KUKA KRL program: EPS_2_251455_MH11A_A_20251003045056.src

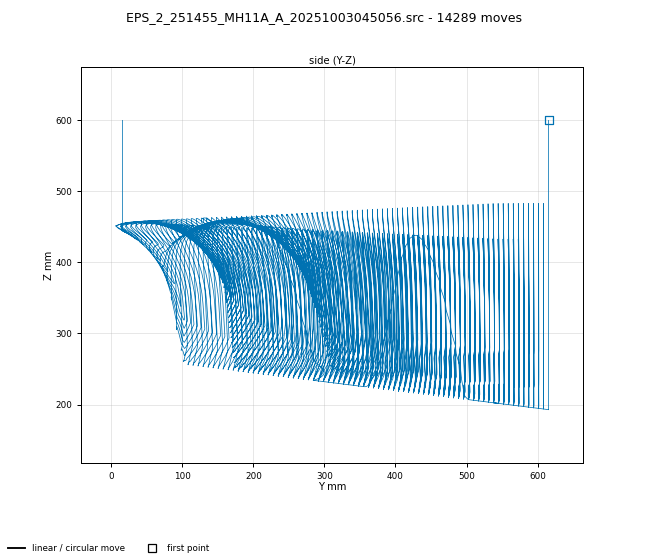
[picture p0: tool path of EPS_2_251455_MH11A_A_20251003045056.src, 14289 of 14291 moves have a stored position in this frame; points joined in program order, loops and branches not executed]
&ACCESS RVP
&REL 4
&COMMENT QRS 19112012
&PARAM EDITMASK = *
DEF PART()
EXT BAS (BAS_COMMAND :IN,REAL :IN )
INT I
BAS (#INITMOV,0 )

;KUKA QRS Post kuka4.cps  Date:22-06-2017 !

File_ID=2867

QRS_PRE_INIT()

;Init var - Until changes are made in qrs_pre_init
Outlet_Square_prg=0
Inlet_1_Square_prg=0
Inlet_2_Square_prg=0
Inlet_3_Square_prg=0
Inlet_4_Square_prg=0
Inlet_5_Square_prg=0

Outlet_1={X 0.000, Y 540.910, Z 382.500, B 0.000, E1 0.000 }
Inlet_1={X 0.000, Y 544.470, Z 332.500, B 0.000, E1 166.000 }
Inlet_2={X 0.000, Y 544.470, Z 332.500, B 0.000, E1 269.000 }
Outlet_1_type=201
Inlet_1_type=201
Inlet_2_type=201
;QRS#1=Sidecore dimensions
;QRS#2=200-8" PVC SDR 35
;QRS#3=200-8" PVC SDR 35
;QRS#4=200-8" PVC SDR 35
;QRS#5=
;QRS#6=
;QRS#7=
;QRS#8=
;QRS#9=12-08 PSX
;QRS#10=12-08 PSX
;QRS#11=12-08 PSX
;QRS#12=
;QRS#13=
;QRS#14=
;QRS#15=
;QRS#16=1220x127x762 2,5'
;QRS#17=EPS Height
;QRS#18=483
;QRS#19=*
;QRS#20= UPDATED VERSION 22-06-2017
;QRS#21=*
Outlet_Square=0100
Inlet_1_Square=0100
Inlet_2_Square=0100
Inlet_3_Square=0
Inlet_4_Square=0
Inlet_5_Square=0
Mill_Square=1
Outlet_Square_Prg=204
Inlet_1_Square_prg=204
Inlet_2_Square_prg=204

QRS_INIT()

$ADVANCE=5

; T1
PTP {E1 173.609,E2 173.609}
PTP {X 0,Y 615.501,A -85,B 0,C 180,E1 173.609,E2 173.609,E3 0,E4 0,E5 0,E6 0}
QRS_SPEED_INIT()
LIN {X 0,Y 615.501,Z 600,A -85,B 0,C 180,E1 173.609,E2 173.609,E3 0,E4 0,E5 0,E6 0} C_VEL
LIN {X 0,Y 615.501,Z 202.87,A -85,B 0,C 180,E1 173.609,E2 173.609} C_VEL
LIN {X 0,Y 615.501,Z 194.691,A -85,B 0,C 180,E1 173.609,E2 173.609} C_VEL
LIN {X 0,Y 615.475,Z 192.691,A -85,B 0,C 180,E1 173.423,E2 173.423} C_VEL
LIN {X 0,Y 615.439,Z 192.695,A -85,B 0,C 180,E1 170.8,E2 170.8} C_VEL
LIN {X 0,Y 615.484,Z 192.701,A -85,B 0,C 180,E1 168.139,E2 168.139} C_VEL
LIN {X 0,Y 615.466,Z 192.69,A -85,B 0,C 180,E1 165.45,E2 165.45} C_VEL
LIN {X 0,Y 615.461,Z 192.69,A -85,B 0,C 180,E1 163.412,E2 163.412} C_VEL
LIN {X 0,Y 615.456,Z 192.69,A -85,B 0,C 180,E1 161.353,E2 161.353} C_VEL
LIN {X 0,Y 615.451,Z 192.691,A -85,B 0,C 180,E1 159.268,E2 159.268} C_VEL
LIN {X 0,Y 615.451,Z 192.692,A -85,B 0,C 180,E1 157.154,E2 157.154} C_VEL
LIN {X 0,Y 615.498,Z 192.699,A -85,B 0,C 180,E1 154.427,E2 154.427} C_VEL
LIN {X 0,Y 615.463,Z 192.689,A -85,B 0,C 180,E1 151.552,E2 151.552} C_VEL
LIN {X 0,Y 615.472,Z 192.697,A -85,B 0,C 180,E1 148.915,E2 148.915} C_VEL
LIN {X 0,Y 615.486,Z 192.685,A -85,B 0,C 180,E1 145.978,E2 145.978} C_VEL
LIN {X 0,Y 615.462,Z 192.689,A -85,B 0,C 180,E1 143.573,E2 143.573} C_VEL
LIN {X 0,Y 615.492,Z 192.699,A -85,B 0,C 180,E1 140.936,E2 140.936} C_VEL
LIN {X 0,Y 615.476,Z 192.686,A -85,B 0,C 180,E1 137.92,E2 137.92} C_VEL
LIN {X 0,Y 615.496,Z 192.699,A -85,B 0,C 180,E1 135.066,E2 135.066} C_VEL
LIN {X 0,Y 615.481,Z 192.684,A -85,B 0,C 180,E1 132.079,E2 132.079} C_VEL
LIN {X 0,Y 615.47,Z 192.691,A -85,B 0,C 180,E1 129.75,E2 129.75} C_VEL
LIN {X 0,Y 615.484,Z 192.693,A -85,B 0,C 180,E1 126.935,E2 126.935} C_VEL
LIN {X 0,Y 615.473,Z 192.688,A -85,B 0,C 180,E1 124.022,E2 124.022} C_VEL
LIN {X 0,Y 615.475,Z 192.815,A -85,B 0,C 180,E1 121.967,E2 121.967} C_VEL
LIN {X 0,Y 615.473,Z 207.433,A -85,B 0,C 180,E1 119.406,E2 119.406} C_VEL
LIN {X 0,Y 615.47,Z 222.393,A -85,B 0,C 180,E1 116.814,E2 116.814} C_VEL
LIN {X 0,Y 615.432,Z 328.155,A -85,B 0,C 180,E1 115.557,E2 115.557} C_VEL
LIN {X 0,Y 615.439,Z 341.34,A -85,B 0,C 180,E1 115.274,E2 115.274} C_VEL
LIN {X 0,Y 615.476,Z 354.247,A -85,B 0,C 180,E1 114.856,E2 114.856} C_VEL
LIN {X 0,Y 615.479,Z 365.558,A -85,B 0,C 180,E1 114.361,E2 114.361} C_VEL
LIN {X 0,Y 615.469,Z 376.031,A -85,B 0,C 180,E1 113.779,E2 113.779} C_VEL
LIN {X 0,Y 615.498,Z 386.868,A -85,B 0,C 180,E1 113.021,E2 113.021} C_VEL
LIN {X 0,Y 615.498,Z 397.085,A -85,B 0,C 180,E1 112.135,E2 112.135} C_VEL
LIN {X 0,Y 615.497,Z 405.273,A -85,B 0,C 180,E1 111.255,E2 111.255} C_VEL
LIN {X 0,Y 615.496,Z 412.557,A -85,B 0,C 180,E1 110.295,E2 110.295} C_VEL
LIN {X 0,Y 615.497,Z 418.434,A -85,B 0,C 180,E1 109.337,E2 109.337} C_VEL
LIN {X 0,Y 615.496,Z 423.553,A -85,B 0,C 180,E1 108.281,E2 108.281} C_VEL
LIN {X 0,Y 615.498,Z 427.265,A -85,B 0,C 180,E1 107.269,E2 107.269} C_VEL
LIN {X 0,Y 615.495,Z 429.552,A -85,B 0,C 180,E1 106.432,E2 106.432} C_VEL
LIN {X 0,Y 615.496,Z 431.625,A -85,B 0,C 180,E1 105.225,E2 105.225} C_VEL
LIN {X 0,Y 615.499,Z 432.387,A -85,B 0,C 180,E1 103.935,E2 103.935} C_VEL
LIN {X 0,Y 615.496,Z 432.102,A -85,B 0,C 180,E1 103.2,E2 103.2} C_VEL
LIN {X 0,Y 615.496,Z 431.442,A -85,B 0,C 180,E1 102.529,E2 102.529} C_VEL
LIN {X 0,Y 615.494,Z 430.377,A -85,B 0,C 180,E1 101.86,E2 101.86} C_VEL
LIN {X 0,Y 615.495,Z 428.034,A -85,B 0,C 180,E1 100.889,E2 100.889} C_VEL
LIN {X 0,Y 615.498,Z 424.523,A -85,B 0,C 180,E1 99.861,E2 99.861} C_VEL
LIN {X 0,Y 615.498,Z 420.016,A -85,B 0,C 180,E1 98.867,E2 98.867} C_VEL
LIN {X 0,Y 615.499,Z 413.193,A -85,B 0,C 180,E1 97.71,E2 97.71} C_VEL
LIN {X 0,Y 615.498,Z 405.966,A -85,B 0,C 180,E1 96.74,E2 96.74} C_VEL
LIN {X 0,Y 615.499,Z 398.311,A -85,B 0,C 180,E1 95.898,E2 95.898} C_VEL
LIN {X 0,Y 615.498,Z 389.248,A -85,B 0,C 180,E1 95.076,E2 95.076} C_VEL
LIN {X 0,Y 615.477,Z 379.211,A -85,B 0,C 180,E1 94.338,E2 94.338} C_VEL
LIN {X 0,Y 615.462,Z 368.138,A -85,B 0,C 180,E1 93.682,E2 93.682} C_VEL
LIN {X 0,Y 615.496,Z 357.647,A -85,B 0,C 180,E1 93.19,E2 93.19} C_VEL
LIN {X 0,Y 615.477,Z 345.076,A -85,B 0,C 180,E1 92.74,E2 92.74} C_VEL
LIN {X 0,Y 615.457,Z 332.551,A -85,B 0,C 180,E1 92.433,E2 92.433} C_VEL
LIN {X 0,Y 615.454,Z 314.913,A -85,B 0,C 180,E1 92.188,E2 92.188} C_VEL
LIN {X 0,Y 615.495,Z 222.43,A -85,B 0,C 180,E1 91.103,E2 91.103} C_VEL
LIN {X 0,Y 615.488,Z 206.621,A -85,B 0,C 180,E1 88.363,E2 88.363} C_VEL
LIN {X 0,Y 615.455,Z 192.693,A -85,B 0,C 180,E1 85.907,E2 85.907} C_VEL
LIN {X 0,Y 615.467,Z 192.688,A -85,B 0,C 180,E1 83.442,E2 83.442} C_VEL
LIN {X 0,Y 615.495,Z 192.696,A -85,B 0,C 180,E1 80.801,E2 80.801} C_VEL
LIN {X 0,Y 615.451,Z 192.695,A -85,B 0,C 180,E1 78.138,E2 78.138} C_VEL
LIN {X 0,Y 615.444,Z 192.695,A -85,B 0,C 180,E1 76.086,E2 76.086} C_VEL
LIN {X 0,Y 615.483,Z 192.688,A -85,B 0,C 180,E1 73.413,E2 73.413} C_VEL
LIN {X 0,Y 615.467,Z 192.698,A -85,B 0,C 180,E1 70.661,E2 70.661} C_VEL
LIN {X 0,Y 615.454,Z 192.697,A -85,B 0,C 180,E1 68.566,E2 68.566} C_VEL
LIN {X 0,Y 615.443,Z 192.693,A -85,B 0,C 180,E1 66.002,E2 66.002} C_VEL
LIN {X 0,Y 615.479,Z 192.692,A -85,B 0,C 180,E1 63.555,E2 63.555} C_VEL
LIN {X 0,Y 615.493,Z 192.697,A -85,B 0,C 180,E1 61.342,E2 61.342} C_VEL
LIN {X 0,Y 615.456,Z 192.698,A -85,B 0,C 180,E1 58.92,E2 58.92} C_VEL
LIN {X 0,Y 615.429,Z 192.697,A -85,B 0,C 180,E1 56.475,E2 56.475} C_VEL
LIN {X 0,Y 615.437,Z 192.695,A -85,B 0,C 180,E1 54.174,E2 54.174} C_VEL
LIN {X 0,Y 615.46,Z 192.695,A -85,B 0,C 180,E1 51.929,E2 51.929} C_VEL
LIN {X 0,Y 615.478,Z 192.7,A -85,B 0,C 180,E1 49.392,E2 49.392} C_VEL
LIN {X 0,Y 615.428,Z 192.699,A -85,B 0,C 180,E1 46.959,E2 46.959} C_VEL
LIN {X 0,Y 615.422,Z 192.699,A -85,B 0,C 180,E1 44.925,E2 44.925} C_VEL
LIN {X 0,Y 615.459,Z 192.698,A -85,B 0,C 180,E1 42.076,E2 42.076} C_VEL
LIN {X 0,Y 615.484,Z 192.701,A -85,B 0,C 180,E1 39.751,E2 39.751} C_VEL
LIN {X 0,Y 615.423,Z 192.7,A -85,B 0,C 180,E1 37.247,E2 37.247} C_VEL
LIN {X 0,Y 615.455,Z 192.7,A -85,B 0,C 180,E1 35.618,E2 35.618} C_VEL
LIN {X 0,Y 615.422,Z 192.699,A -85,B 0,C 180,E1 33.241,E2 33.241} C_VEL
LIN {X 0,Y 615.418,Z 192.699,A -85,B 0,C 180,E1 30.924,E2 30.924} C_VEL
LIN {X 0,Y 615.457,Z 192.699,A -85,B 0,C 180,E1 28.444,E2 28.444} C_VEL
LIN {X 0,Y 615.439,Z 192.696,A -85,B 0,C 180,E1 25.558,E2 25.558} C_VEL
LIN {X 0,Y 615.438,Z 192.696,A -85,B 0,C 180,E1 23.559,E2 23.559} C_VEL
LIN {X 0,Y 615.431,Z 192.696,A -85,B 0,C 180,E1 21.434,E2 21.434} C_VEL
LIN {X 0,Y 615.439,Z 192.798,A -85,B 0,C 180,E1 18.972,E2 18.972} C_VEL
LIN {X 0,Y 615.49,Z 208.798,A -85,B 0,C 180,E1 16.168,E2 16.168} C_VEL
LIN {X 0,Y 615.482,Z 222.406,A -85,B 0,C 180,E1 13.811,E2 13.811} C_VEL
LIN {X 0,Y 615.482,Z 329.594,A -85,B 0,C 180,E1 12.53,E2 12.53} C_VEL
LIN {X 0,Y 615.496,Z 342.645,A -85,B 0,C 180,E1 12.237,E2 12.237} C_VEL
LIN {X 0,Y 615.494,Z 355.228,A -85,B 0,C 180,E1 11.819,E2 11.819} C_VEL
LIN {X 0,Y 615.465,Z 367.214,A -85,B 0,C 180,E1 11.277,E2 11.277} C_VEL
LIN {X 0,Y 615.476,Z 378.576,A -85,B 0,C 180,E1 10.614,E2 10.614} C_VEL
LIN {X 0,Y 615.499,Z 388.888,A -85,B 0,C 180,E1 9.862,E2 9.862} C_VEL
LIN {X 0,Y 615.497,Z 398.107,A -85,B 0,C 180,E1 9.033,E2 9.033} C_VEL
LIN {X 0,Y 615.498,Z 407.028,A -85,B 0,C 180,E1 8.041,E2 8.041} C_VEL
LIN {X 0,Y 615.497,Z 414.162,A -85,B 0,C 180,E1 7.057,E2 7.057} C_VEL
LIN {X 0,Y 615.498,Z 419.032,A -85,B 0,C 180,E1 6.228,E2 6.228} C_VEL
LIN {X 0,Y 615.495,Z 423.722,A -85,B 0,C 180,E1 5.241,E2 5.241} C_VEL
LIN {X 0,Y 615.496,Z 427.306,A -85,B 0,C 180,E1 4.257,E2 4.257} C_VEL
LIN {X 0,Y 615.496,Z 429.894,A -85,B 0,C 180,E1 3.273,E2 3.273} C_VEL
LIN {X 0,Y 615.497,Z 431.108,A -85,B 0,C 180,E1 2.618,E2 2.618} C_VEL
LIN {X 0,Y 615.496,Z 431.923,A -85,B 0,C 180,E1 1.963,E2 1.963} C_VEL
LIN {X 0,Y 615.495,Z 432.323,A -85,B 0,C 180,E1 0.654,E2 0.654} C_VEL
LIN {X 0,Y 615.495,Z 431.962,A -85,B 0,C 180,E1 0,E2 0} C_VEL
LIN {X 0,Y 615.496,Z 431.198,A -85,B 0,C 180,E1 -0.654,E2 -0.654} C_VEL
LIN {X 0,Y 615.499,Z 428.43,A -85,B 0,C 180,E1 -1.963,E2 -1.963} C_VEL
LIN {X 0,Y 615.496,Z 425.246,A -85,B 0,C 180,E1 -2.945,E2 -2.945} C_VEL
LIN {X 0,Y 615.495,Z 421.016,A -85,B 0,C 180,E1 -3.928,E2 -3.928} C_VEL
LIN {X 0,Y 615.497,Z 414.61,A -85,B 0,C 180,E1 -5.077,E2 -5.077} C_VEL
LIN {X 0,Y 615.497,Z 407.586,A -85,B 0,C 180,E1 -6.063,E2 -6.063} C_VEL
LIN {X 0,Y 615.498,Z 398.755,A -85,B 0,C 180,E1 -7.057,E2 -7.057} C_VEL
LIN {X 0,Y 615.497,Z 389.831,A -85,B 0,C 180,E1 -7.875,E2 -7.875} C_VEL
LIN {X 0,Y 615.489,Z 379.866,A -85,B 0,C 180,E1 -8.619,E2 -8.619} C_VEL
LIN {X 0,Y 615.492,Z 368.809,A -85,B 0,C 180,E1 -9.281,E2 -9.281} C_VEL
LIN {X 0,Y 615.489,Z 356.416,A -85,B 0,C 180,E1 -9.862,E2 -9.862} C_VEL
LIN {X 0,Y 615.452,Z 344.471,A -85,B 0,C 180,E1 -10.278,E2 -10.278} C_VEL
LIN {X 0,Y 615.446,Z 331.21,A -85,B 0,C 180,E1 -10.592,E2 -10.592} C_VEL
LIN {X 0,Y 615.455,Z 309.997,A -85,B 0,C 180,E1 -10.87,E2 -10.87} C_VEL
LIN {X 0,Y 615.449,Z 222.404,A -85,B 0,C 180,E1 -11.903,E2 -11.903} C_VEL
LIN {X 0,Y 615.447,Z 208.959,A -85,B 0,C 180,E1 -14.232,E2 -14.232} C_VEL
LIN {X 0,Y 615.489,Z 193.058,A -85,B 0,C 180,E1 -17.014,E2 -17.014} C_VEL
LIN {X 0,Y 615.488,Z 192.686,A -85,B 0,C 180,E1 -17.099,E2 -17.099} C_VEL
LIN {X 0,Y 615.483,Z 192.684,A -85,B 0,C 180,E1 -19.338,E2 -19.338} C_VEL
LIN {X 0,Y 615.472,Z 192.696,A -85,B 0,C 180,E1 -22.137,E2 -22.137} C_VEL
LIN {X 0,Y 615.495,Z 192.684,A -85,B 0,C 180,E1 -24.991,E2 -24.991} C_VEL
LIN {X 0,Y 615.486,Z 192.683,A -85,B 0,C 180,E1 -27.177,E2 -27.177} C_VEL
LIN {X 0,Y 615.463,Z 192.693,A -85,B 0,C 180,E1 -29.79,E2 -29.79} C_VEL
LIN {X 0,Y 615.49,Z 192.696,A -85,B 0,C 180,E1 -32.457,E2 -32.457} C_VEL
LIN {X 0,Y 615.493,Z 192.685,A -85,B 0,C 180,E1 -34.815,E2 -34.815} C_VEL
LIN {X 0,Y 615.468,Z 192.687,A -85,B 0,C 180,E1 -37.244,E2 -37.244} C_VEL
LIN {X 0,Y 615.491,Z 192.699,A -85,B 0,C 180,E1 -40.089,E2 -40.089} C_VEL
LIN {X 0,Y 615.475,Z 192.685,A -85,B 0,C 180,E1 -43.045,E2 -43.045} C_VEL
LIN {X 0,Y 615.476,Z 192.697,A -85,B 0,C 180,E1 -45.849,E2 -45.849} C_VEL
LIN {X 0,Y 615.493,Z 192.687,A -85,B 0,C 180,E1 -48.526,E2 -48.526} C_VEL
LIN {X 0,Y 615.463,Z 192.688,A -85,B 0,C 180,E1 -51.093,E2 -51.093} C_VEL
LIN {X 0,Y 615.465,Z 192.695,A -85,B 0,C 180,E1 -53.573,E2 -53.573} C_VEL
LIN {X 0,Y 615.495,Z 192.685,A -85,B 0,C 180,E1 -56.465,E2 -56.465} C_VEL
LIN {X 0,Y 615.459,Z 192.69,A -85,B 0,C 180,E1 -59.078,E2 -59.078} C_VEL
LIN {X 0,Y 615.47,Z 192.696,A -85,B 0,C 180,E1 -61.553,E2 -61.553} C_VEL
LIN {X 0,Y 615.498,Z 192.683,A -85,B 0,C 180,E1 -64.43,E2 -64.43} C_VEL
LIN {X 0,Y 615.456,Z 192.818,A -85,B 0,C 180,E1 -67.065,E2 -67.065} C_VEL
LIN {X 0,Y 615.471,Z 212.766,A -85,B 0,C 180,E1 -69.706,E2 -69.706} C_VEL
LIN {X 0,Y 615.477,Z 234.665,A -85,B 0,C 180,E1 -72.557,E2 -72.557} C_VEL
LIN {X 0,Y 615.471,Z 255.886,A -85,B 0,C 180,E1 -75.281,E2 -75.281} C_VEL
LIN {X 0,Y 615.452,Z 270.295,A -85,B 0,C 180,E1 -77.112,E2 -77.112} C_VEL
LIN {X 0,Y 615.483,Z 378.793,A -85,B 0,C 180,E1 -78.41,E2 -78.41} C_VEL
LIN {X 0,Y 615.474,Z 391.321,A -85,B 0,C 180,E1 -78.681,E2 -78.681} C_VEL
LIN {X 0,Y 615.487,Z 404.628,A -85,B 0,C 180,E1 -79.113,E2 -79.113} C_VEL
LIN {X 0,Y 615.479,Z 416.465,A -85,B 0,C 180,E1 -79.639,E2 -79.639} C_VEL
LIN {X 0,Y 615.496,Z 427.983,A -85,B 0,C 180,E1 -80.303,E2 -80.303} C_VEL
LIN {X 0,Y 615.499,Z 438.332,A -85,B 0,C 180,E1 -81.049,E2 -81.049} C_VEL
LIN {X 0,Y 615.497,Z 446.804,A -85,B 0,C 180,E1 -81.793,E2 -81.793} C_VEL
LIN {X 0,Y 615.498,Z 454.6,A -85,B 0,C 180,E1 -82.619,E2 -82.619} C_VEL
LIN {X 0,Y 615.496,Z 462.198,A -85,B 0,C 180,E1 -83.607,E2 -83.607} C_VEL
LIN {X 0,Y 615.498,Z 469.201,A -85,B 0,C 180,E1 -84.758,E2 -84.758} C_VEL
LIN {X 0,Y 615.494,Z 473.848,A -85,B 0,C 180,E1 -85.743,E2 -85.743} C_VEL
LIN {X 0,Y 615.494,Z 477.396,A -85,B 0,C 180,E1 -86.726,E2 -86.726} C_VEL
LIN {X 0,Y 615.497,Z 479.231,A -85,B 0,C 180,E1 -87.381,E2 -87.381} C_VEL
LIN {X 0,Y 615.5,Z 480.606,A -85,B 0,C 180,E1 -88.036,E2 -88.036} C_VEL
LIN {X 0,Y 615.496,Z 482.173,A -85,B 0,C 180,E1 -89.345,E2 -89.345} C_VEL
LIN {X 0,Y 615.494,Z 482.389,A -85,B 0,C 180,E1 -89.999,E2 -89.999} C_VEL
LIN {X 0,Y 615.495,Z 481.581,A -85,B 0,C 180,E1 -91.308,E2 -91.308} C_VEL
LIN {X 0,Y 615.5,Z 480.609,A -85,B 0,C 180,E1 -91.962,E2 -91.962} C_VEL
LIN {X 0,Y 615.497,Z 479.235,A -85,B 0,C 180,E1 -92.617,E2 -92.617} C_VEL
LIN {X 0,Y 615.496,Z 476.352,A -85,B 0,C 180,E1 -93.6,E2 -93.6} C_VEL
LIN {X 0,Y 615.498,Z 472.445,A -85,B 0,C 180,E1 -94.584,E2 -94.584} C_VEL
LIN {X 0,Y 615.499,Z 467.409,A -85,B 0,C 180,E1 -95.569,E2 -95.569} C_VEL
LIN {X 0,Y 615.497,Z 460.869,A -85,B 0,C 180,E1 -96.583,E2 -96.583} C_VEL
LIN {X 0,Y 615.497,Z 453.14,A -85,B 0,C 180,E1 -97.545,E2 -97.545} C_VEL
LIN {X 0,Y 615.498,Z 445.053,A -85,B 0,C 180,E1 -98.37,E2 -98.37} C_VEL
LIN {X 0,Y 615.499,Z 435.178,A -85,B 0,C 180,E1 -99.198,E2 -99.198} C_VEL
LIN {X 0,Y 615.492,Z 423.994,A -85,B 0,C 180,E1 -99.944,E2 -99.944} C_VEL
LIN {X 0,Y 615.483,Z 413.039,A -85,B 0,C 180,E1 -100.526,E2 -100.526} C_VEL
LIN {X 0,Y 615.478,Z 400.507,A -85,B 0,C 180,E1 -101.04,E2 -101.04} C_VEL
LIN {X 0,Y 615.475,Z 388.102,A -85,B 0,C 180,E1 -101.401,E2 -101.401} C_VEL
LIN {X 0,Y 615.487,Z 374.523,A -85,B 0,C 180,E1 -101.651,E2 -101.651} C_VEL
LIN {X 0,Y 615.452,Z 270.307,A -85,B 0,C 180,E1 -102.886,E2 -102.886} C_VEL
LIN {X 0,Y 615.498,Z 247.939,A -85,B 0,C 180,E1 -105.734,E2 -105.734} C_VEL
LIN {X 0,Y 615.452,Z 225.786,A -85,B 0,C 180,E1 -108.594,E2 -108.594} C_VEL
LIN {X 0,Y 615.484,Z 205.459,A -85,B 0,C 180,E1 -111.256,E2 -111.256} C_VEL
LIN {X 0,Y 615.456,Z 192.691,A -85,B 0,C 180,E1 -112.978,E2 -112.978} C_VEL
LIN {X 0,Y 615.493,Z 192.689,A -85,B 0,C 180,E1 -115.715,E2 -115.715} C_VEL
LIN {X 0,Y 615.453,Z 192.694,A -85,B 0,C 180,E1 -118.659,E2 -118.659} C_VEL
LIN {X 0,Y 615.461,Z 192.689,A -85,B 0,C 180,E1 -121.081,E2 -121.081} C_VEL
LIN {X 0,Y 615.481,Z 192.7,A -85,B 0,C 180,E1 -124.021,E2 -124.021} C_VEL
LIN {X 0,Y 615.448,Z 192.695,A -85,B 0,C 180,E1 -126.426,E2 -126.426} C_VEL
LIN {X 0,Y 615.466,Z 192.69,A -85,B 0,C 180,E1 -129.059,E2 -129.059} C_VEL
LIN {X 0,Y 615.494,Z 192.694,A -85,B 0,C 180,E1 -131.472,E2 -131.472} C_VEL
LIN {X 0,Y 615.445,Z 192.697,A -85,B 0,C 180,E1 -134.152,E2 -134.152} C_VEL
LIN {X 0,Y 615.467,Z 192.692,A -85,B 0,C 180,E1 -136.953,E2 -136.953} C_VEL
LIN {X 0,Y 615.446,Z 192.698,A -85,B 0,C 180,E1 -139.914,E2 -139.914} C_VEL
LIN {X 0,Y 615.434,Z 192.698,A -85,B 0,C 180,E1 -141.993,E2 -141.993} C_VEL
LIN {X 0,Y 615.432,Z 192.696,A -85,B 0,C 180,E1 -144.38,E2 -144.38} C_VEL
LIN {X 0,Y 615.461,Z 192.695,A -85,B 0,C 180,E1 -146.762,E2 -146.762} C_VEL
LIN {X 0,Y 615.492,Z 192.699,A -85,B 0,C 180,E1 -149.08,E2 -149.08} C_VEL
LIN {X 0,Y 615.442,Z 192.699,A -85,B 0,C 180,E1 -151.556,E2 -151.556} C_VEL
LIN {X 0,Y 615.435,Z 192.7,A -85,B 0,C 180,E1 -153.553,E2 -153.553} C_VEL
LIN {X 0,Y 615.421,Z 192.699,A -85,B 0,C 180,E1 -155.725,E2 -155.725} C_VEL
LIN {X 0,Y 615.413,Z 192.7,A -85,B 0,C 180,E1 -157.861,E2 -157.861} C_VEL
LIN {X 0,Y 615.474,Z 192.7,A -85,B 0,C 180,E1 -160.662,E2 -160.662} C_VEL
LIN {X 0,Y 615.424,Z 192.7,A -85,B 0,C 180,E1 -163.412,E2 -163.412} C_VEL
LIN {X 0,Y 615.422,Z 192.699,A -85,B 0,C 180,E1 -165.449,E2 -165.449} C_VEL
LIN {X 0,Y 615.42,Z 192.699,A -85,B 0,C 180,E1 -167.469,E2 -167.469} C_VEL
LIN {X 0,Y 615.422,Z 192.698,A -85,B 0,C 180,E1 -169.472,E2 -169.472} C_VEL
LIN {X 0,Y 615.423,Z 192.698,A -85,B 0,C 180,E1 -171.463,E2 -171.463} C_VEL
LIN {X 0,Y 615.454,Z 192.699,A -85,B 0,C 180,E1 -174.101,E2 -174.101} C_VEL
LIN {X 0,Y 615.473,Z 192.694,A -85,B 0,C 180,E1 -176.727,E2 -176.727} C_VEL
LIN {X 0,Y 615.43,Z 192.696,A -85,B 0,C 180,E1 -179.346,E2 -179.346} C_VEL
LIN {X 0,Y 615.467,Z 192.699,A -85,B 0,C 180,E1 -181.963,E2 -181.963} C_VEL
LIN {X 0,Y 615.478,Z 192.691,A -85,B 0,C 180,E1 -184.585,E2 -184.585} C_VEL
LIN {X 0,Y 615.475,Z 192.691,A -85,B 0,C 180,E1 -186.577,E2 -186.577} C_VEL
LIN {X 0,Y 614.772,Z 192.839,A -85,B 0,C 180,E1 -187.123,E2 -187.123} C_VEL
LIN {X 0,Y 611.916,Z 193.266,A -85,B 0,C 180,E1 -188.009,E2 -188.009} C_VEL
LIN {X 0,Y 609.53,Z 193.569,A -85,B 0,C 180,E1 -188.721,E2 -188.721} C_VEL
LIN {X 0,Y 608.51,Z 193.683,A -85,B 0,C 180,E1 -189.271,E2 -189.271} C_VEL
LIN {X 0,Y 608.429,Z 193.693,A -85,B 0,C 180,E1 -189.457,E2 -189.457} C_VEL
LIN {X 0,Y 608.456,Z 193.696,A -85,B 0,C 180,E1 -192,E2 -192} C_VEL
LIN {X 0,Y 608.453,Z 193.688,A -85,B 0,C 180,E1 -194.721,E2 -194.721} C_VEL
LIN {X 0,Y 608.434,Z 193.695,A -85,B 0,C 180,E1 -197.477,E2 -197.477} C_VEL
LIN {X 0,Y 608.455,Z 193.689,A -85,B 0,C 180,E1 -200.275,E2 -200.275} C_VEL
LIN {X 0,Y 608.452,Z 193.688,A -85,B 0,C 180,E1 -202.477,E2 -202.477} C_VEL
LIN {X 0,Y 608.437,Z 193.689,A -85,B 0,C 180,E1 -204.572,E2 -204.572} C_VEL
LIN {X 0,Y 608.463,Z 193.692,A -85,B 0,C 180,E1 -207.206,E2 -207.206} C_VEL
LIN {X 0,Y 608.469,Z 193.687,A -85,B 0,C 180,E1 -209.974,E2 -209.974} C_VEL
LIN {X 0,Y 608.439,Z 193.69,A -85,B 0,C 180,E1 -212.521,E2 -212.521} C_VEL
LIN {X 0,Y 608.433,Z 193.694,A -85,B 0,C 180,E1 -214.905,E2 -214.905} C_VEL
LIN {X 0,Y 608.476,Z 193.695,A -85,B 0,C 180,E1 -217.161,E2 -217.161} C_VEL
LIN {X 0,Y 608.477,Z 193.69,A -85,B 0,C 180,E1 -219.44,E2 -219.44} C_VEL
LIN {X 0,Y 608.438,Z 193.69,A -85,B 0,C 180,E1 -222.333,E2 -222.333} C_VEL
LIN {X 0,Y 608.46,Z 193.694,A -85,B 0,C 180,E1 -224.796,E2 -224.796} C_VEL
LIN {X 0,Y 608.467,Z 193.686,A -85,B 0,C 180,E1 -227.666,E2 -227.666} C_VEL
LIN {X 0,Y 608.446,Z 193.697,A -85,B 0,C 180,E1 -230.706,E2 -230.706} C_VEL
LIN {X 0,Y 608.455,Z 193.692,A -85,B 0,C 180,E1 -233.086,E2 -233.086} C_VEL
LIN {X 0,Y 608.465,Z 193.686,A -85,B 0,C 180,E1 -235.532,E2 -235.532} C_VEL
LIN {X 0,Y 608.479,Z 193.809,A -85,B 0,C 180,E1 -237.981,E2 -237.981} C_VEL
LIN {X 0,Y 608.464,Z 208.651,A -85,B 0,C 180,E1 -240.602,E2 -240.602} C_VEL
LIN {X 0,Y 608.442,Z 222.619,A -85,B 0,C 180,E1 -243.039,E2 -243.039} C_VEL
LIN {X 0,Y 608.499,Z 329.351,A -85,B 0,C 180,E1 -244.328,E2 -244.328} C_VEL
LIN {X 0,Y 608.475,Z 342.727,A -85,B 0,C 180,E1 -244.63,E2 -244.63} C_VEL
LIN {X 0,Y 608.523,Z 355.714,A -85,B 0,C 180,E1 -245.069,E2 -245.069} C_VEL
LIN {X 0,Y 608.498,Z 367.699,A -85,B 0,C 180,E1 -245.621,E2 -245.621} C_VEL
LIN {X 0,Y 608.481,Z 379.741,A -85,B 0,C 180,E1 -246.337,E2 -246.337} C_VEL
LIN {X 0,Y 608.491,Z 390.515,A -85,B 0,C 180,E1 -247.148,E2 -247.148} C_VEL
LIN {X 0,Y 608.456,Z 399.194,A -85,B 0,C 180,E1 -247.952,E2 -247.952} C_VEL
LIN {X 0,Y 608.449,Z 407.117,A -85,B 0,C 180,E1 -248.842,E2 -248.842} C_VEL
LIN {X 0,Y 608.438,Z 414.789,A -85,B 0,C 180,E1 -249.902,E2 -249.902} C_VEL
LIN {X 0,Y 608.44,Z 419.887,A -85,B 0,C 180,E1 -250.781,E2 -250.781} C_VEL
LIN {X 0,Y 608.43,Z 424.752,A -85,B 0,C 180,E1 -251.828,E2 -251.828} C_VEL
LIN {X 0,Y 608.453,Z 428.39,A -85,B 0,C 180,E1 -252.871,E2 -252.871} C_VEL
LIN {X 0,Y 608.434,Z 430.925,A -85,B 0,C 180,E1 -253.906,E2 -253.906} C_VEL
LIN {X 0,Y 608.42,Z 432.034,A -85,B 0,C 180,E1 -254.594,E2 -254.594} C_VEL
LIN {X 0,Y 608.418,Z 432.71,A -85,B 0,C 180,E1 -255.279,E2 -255.279} C_VEL
LIN {X 0,Y 608.445,Z 432.994,A -85,B 0,C 180,E1 -255.995,E2 -255.995} C_VEL
LIN {X 0,Y 608.439,Z 432.828,A -85,B 0,C 180,E1 -256.644,E2 -256.644} C_VEL
LIN {X 0,Y 608.439,Z 431.251,A -85,B 0,C 180,E1 -258.001,E2 -258.001} C_VEL
LIN {X 0,Y 608.423,Z 428.806,A -85,B 0,C 180,E1 -259.07,E2 -259.07} C_VEL
LIN {X 0,Y 608.437,Z 425.661,A -85,B 0,C 180,E1 -260.023,E2 -260.023} C_VEL
LIN {X 0,Y 608.448,Z 421.293,A -85,B 0,C 180,E1 -261.03,E2 -261.03} C_VEL
LIN {X 0,Y 608.439,Z 415.738,A -85,B 0,C 180,E1 -262.033,E2 -262.033} C_VEL
LIN {X 0,Y 608.466,Z 408.822,A -85,B 0,C 180,E1 -263.035,E2 -263.035} C_VEL
LIN {X 0,Y 608.455,Z 400.205,A -85,B 0,C 180,E1 -264.034,E2 -264.034} C_VEL
LIN {X 0,Y 608.483,Z 391.401,A -85,B 0,C 180,E1 -264.865,E2 -264.865} C_VEL
LIN {X 0,Y 608.492,Z 380.606,A -85,B 0,C 180,E1 -265.695,E2 -265.695} C_VEL
LIN {X 0,Y 608.483,Z 369.765,A -85,B 0,C 180,E1 -266.359,E2 -266.359} C_VEL
LIN {X 0,Y 608.513,Z 357.695,A -85,B 0,C 180,E1 -266.939,E2 -266.939} C_VEL
LIN {X 0,Y 608.509,Z 345.045,A -85,B 0,C 180,E1 -267.394,E2 -267.394} C_VEL
LIN {X 0,Y 608.513,Z 332.437,A -85,B 0,C 180,E1 -267.705,E2 -267.705} C_VEL
LIN {X 0,Y 608.512,Z 314.675,A -85,B 0,C 180,E1 -267.953,E2 -267.953} C_VEL
LIN {X 0,Y 608.468,Z 222.627,A -85,B 0,C 180,E1 -269.049,E2 -269.049} C_VEL
LIN {X 0,Y 608.482,Z 207.696,A -85,B 0,C 180,E1 -271.655,E2 -271.655} C_VEL
LIN {X 0,Y 608.434,Z 193.692,A -85,B 0,C 180,E1 -274.141,E2 -274.141} C_VEL
LIN {X 0,Y 608.443,Z 193.689,A -85,B 0,C 180,E1 -276.634,E2 -276.634} C_VEL
LIN {X 0,Y 608.472,Z 193.695,A -85,B 0,C 180,E1 -279.306,E2 -279.306} C_VEL
LIN {X 0,Y 608.436,Z 193.691,A -85,B 0,C 180,E1 -282.001,E2 -282.001} C_VEL
LIN {X 0,Y 608.439,Z 193.692,A -85,B 0,C 180,E1 -284.722,E2 -284.722} C_VEL
LIN {X 0,Y 608.437,Z 193.694,A -85,B 0,C 180,E1 -287.478,E2 -287.478} C_VEL
LIN {X 0,Y 608.429,Z 193.693,A -85,B 0,C 180,E1 -289.572,E2 -289.572} C_VEL
LIN {X 0,Y 608.438,Z 193.69,A -85,B 0,C 180,E1 -291.693,E2 -291.693} C_VEL
LIN {X 0,Y 608.442,Z 193.694,A -85,B 0,C 180,E1 -294.572,E2 -294.572} C_VEL
LIN {X 0,Y 608.422,Z 193.693,A -85,B 0,C 180,E1 -297.52,E2 -297.52} C_VEL
LIN {X 0,Y 608.426,Z 193.691,A -85,B 0,C 180,E1 -299.964,E2 -299.964} C_VEL
LIN {X 0,Y 608.467,Z 193.693,A -85,B 0,C 180,E1 -302.522,E2 -302.522} C_VEL
LIN {X 0,Y 608.409,Z 193.694,A -85,B 0,C 180,E1 -305.281,E2 -305.281} C_VEL
LIN {X 0,Y 608.445,Z 193.694,A -85,B 0,C 180,E1 -308.237,E2 -308.237} C_VEL
LIN {X 0,Y 608.44,Z 193.697,A -85,B 0,C 180,E1 -310.327,E2 -310.327} C_VEL
LIN {X 0,Y 608.403,Z 193.696,A -85,B 0,C 180,E1 -312.965,E2 -312.965} C_VEL
LIN {X 0,Y 608.401,Z 193.694,A -85,B 0,C 180,E1 -315.198,E2 -315.198} C_VEL
LIN {X 0,Y 608.439,Z 193.694,A -85,B 0,C 180,E1 -317.936,E2 -317.936} C_VEL
LIN {X 0,Y 608.408,Z 193.696,A -85,B 0,C 180,E1 -320.711,E2 -320.711} C_VEL
LIN {X 0,Y 608.382,Z 193.696,A -85,B 0,C 180,E1 -323.079,E2 -323.079} C_VEL
LIN {X 0,Y 608.426,Z 193.694,A -85,B 0,C 180,E1 -325.528,E2 -325.528} C_VEL
LIN {X 0,Y 608.441,Z 193.699,A -85,B 0,C 180,E1 -327.904,E2 -327.904} C_VEL
LIN {X 0,Y 608.455,Z 193.693,A -85,B 0,C 180,E1 -330.219,E2 -330.219} C_VEL
LIN {X 0,Y 608.408,Z 193.693,A -85,B 0,C 180,E1 -332.807,E2 -332.807} C_VEL
LIN {X 0,Y 608.433,Z 193.695,A -85,B 0,C 180,E1 -335.428,E2 -335.428} C_VEL
LIN {X 0,Y 608.44,Z 193.691,A -85,B 0,C 180,E1 -338.307,E2 -338.307} C_VEL
LIN {X 0,Y 608.45,Z 193.793,A -85,B 0,C 180,E1 -340.977,E2 -340.977} C_VEL
LIN {X 0,Y 608.465,Z 210.386,A -85,B 0,C 180,E1 -343.906,E2 -343.906} C_VEL
LIN {X 0,Y 608.455,Z 222.56,A -85,B 0,C 180,E1 -346.029,E2 -346.029} C_VEL
LIN {X 0,Y 608.565,Z 237.122,A -85,B 0,C 180,E1 -346.22,E2 -346.22} C_VEL
LIN {X 0,Y 608.534,Z 329.103,A -85,B 0,C 180,E1 -347.324,E2 -347.324} C_VEL
LIN {X 0,Y 608.552,Z 342.361,A -85,B 0,C 180,E1 -347.621,E2 -347.621} C_VEL
LIN {X 0,Y 608.529,Z 355.057,A -85,B 0,C 180,E1 -348.044,E2 -348.044} C_VEL
LIN {X 0,Y 608.493,Z 367.164,A -85,B 0,C 180,E1 -348.592,E2 -348.592} C_VEL
LIN {X 0,Y 608.469,Z 378.903,A -85,B 0,C 180,E1 -349.282,E2 -349.282} C_VEL
LIN {X 0,Y 608.473,Z 388.998,A -85,B 0,C 180,E1 -350.023,E2 -350.023} C_VEL
LIN {X 0,Y 608.471,Z 398.31,A -85,B 0,C 180,E1 -350.862,E2 -350.862} C_VEL
LIN {X 0,Y 608.463,Z 407.31,A -85,B 0,C 180,E1 -351.866,E2 -351.866} C_VEL
LIN {X 0,Y 608.466,Z 414.558,A -85,B 0,C 180,E1 -352.867,E2 -352.867} C_VEL
LIN {X 0,Y 608.445,Z 420.161,A -85,B 0,C 180,E1 -353.832,E2 -353.832} C_VEL
LIN {X 0,Y 608.44,Z 424.193,A -85,B 0,C 180,E1 -354.698,E2 -354.698} C_VEL
LIN {X 0,Y 608.441,Z 427.826,A -85,B 0,C 180,E1 -355.694,E2 -355.694} C_VEL
LIN {X 0,Y 608.424,Z 430.454,A -85,B 0,C 180,E1 -356.689,E2 -356.689} C_VEL
LIN {X 0,Y 608.425,Z 431.688,A -85,B 0,C 180,E1 -357.352,E2 -357.352} C_VEL
LIN {X 0,Y 608.441,Z 432.52,A -85,B 0,C 180,E1 -358.014,E2 -358.014} C_VEL
LIN {X 0,Y 608.438,Z 432.937,A -85,B 0,C 180,E1 -359.338,E2 -359.338} C_VEL
LIN {X 0,Y 608.435,Z 432.578,A -85,B 0,C 180,E1 -360,E2 -360} C_VEL
LIN {X 0,Y 608.439,Z 431.815,A -85,B 0,C 180,E1 -360.662,E2 -360.662} C_VEL
LIN {X 0,Y 608.449,Z 430.622,A -85,B 0,C 180,E1 -361.324,E2 -361.324} C_VEL
LIN {X 0,Y 608.45,Z 428.079,A -85,B 0,C 180,E1 -362.317,E2 -362.317} C_VEL
LIN {X 0,Y 608.43,Z 424.542,A -85,B 0,C 180,E1 -363.311,E2 -363.311} C_VEL
LIN {X 0,Y 608.441,Z 419.906,A -85,B 0,C 180,E1 -364.306,E2 -364.306} C_VEL
LIN {X 0,Y 608.462,Z 412.91,A -85,B 0,C 180,E1 -365.468,E2 -365.468} C_VEL
LIN {X 0,Y 608.469,Z 405.038,A -85,B 0,C 180,E1 -366.502,E2 -366.502} C_VEL
LIN {X 0,Y 608.472,Z 395.838,A -85,B 0,C 180,E1 -367.466,E2 -367.466} C_VEL
LIN {X 0,Y 608.496,Z 386.04,A -85,B 0,C 180,E1 -368.301,E2 -368.301} C_VEL
LIN {X 0,Y 608.502,Z 375.033,A -85,B 0,C 180,E1 -369.054,E2 -369.054} C_VEL
LIN {X 0,Y 608.501,Z 364.275,A -85,B 0,C 180,E1 -369.641,E2 -369.641} C_VEL
LIN {X 0,Y 608.508,Z 352.459,A -85,B 0,C 180,E1 -370.144,E2 -370.144} C_VEL
LIN {X 0,Y 608.493,Z 339.671,A -85,B 0,C 180,E1 -370.544,E2 -370.544} C_VEL
LIN {X 0,Y 608.506,Z 327.262,A -85,B 0,C 180,E1 -370.795,E2 -370.795} C_VEL
LIN {X 0,Y 608.44,Z 222.799,A -85,B 0,C 180,E1 -372.042,E2 -372.042} C_VEL
LIN {X 0,Y 608.476,Z 207.326,A -85,B 0,C 180,E1 -374.72,E2 -374.72} C_VEL
LIN {X 0,Y 608.461,Z 193.688,A -85,B 0,C 180,E1 -377.151,E2 -377.151} C_VEL
LIN {X 0,Y 608.444,Z 193.689,A -85,B 0,C 180,E1 -379.571,E2 -379.571} C_VEL
LIN {X 0,Y 608.483,Z 193.694,A -85,B 0,C 180,E1 -382.405,E2 -382.405} C_VEL
LIN {X 0,Y 608.442,Z 193.689,A -85,B 0,C 180,E1 -385.301,E2 -385.301} C_VEL
LIN {X 0,Y 608.443,Z 193.689,A -85,B 0,C 180,E1 -387.518,E2 -387.518} C_VEL
LIN {X 0,Y 608.453,Z 193.692,A -85,B 0,C 180,E1 -389.968,E2 -389.968} C_VEL
LIN {X 0,Y 608.454,Z 193.689,A -85,B 0,C 180,E1 -392.88,E2 -392.88} C_VEL
LIN {X 0,Y 608.433,Z 193.69,A -85,B 0,C 180,E1 -395.278,E2 -395.278} C_VEL
LIN {X 0,Y 608.462,Z 193.69,A -85,B 0,C 180,E1 -397.747,E2 -397.747} C_VEL
LIN {X 0,Y 608.455,Z 193.695,A -85,B 0,C 180,E1 -400.329,E2 -400.329} C_VEL
LIN {X 0,Y 608.443,Z 193.689,A -85,B 0,C 180,E1 -402.961,E2 -402.961} C_VEL
LIN {X 0,Y 608.447,Z 193.693,A -85,B 0,C 180,E1 -405.737,E2 -405.737} C_VEL
LIN {X 0,Y 608.46,Z 193.695,A -85,B 0,C 180,E1 -407.938,E2 -407.938} C_VEL
LIN {X 0,Y 608.44,Z 193.69,A -85,B 0,C 180,E1 -410.706,E2 -410.706} C_VEL
LIN {X 0,Y 608.434,Z 193.69,A -85,B 0,C 180,E1 -413.083,E2 -413.083} C_VEL
LIN {X 0,Y 608.456,Z 193.691,A -85,B 0,C 180,E1 -415.529,E2 -415.529} C_VEL
LIN {X 0,Y 608.463,Z 193.697,A -85,B 0,C 180,E1 -417.905,E2 -417.905} C_VEL
LIN {X 0,Y 608.473,Z 193.69,A -85,B 0,C 180,E1 -420.22,E2 -420.22} C_VEL
LIN {X 0,Y 608.463,Z 193.686,A -85,B 0,C 180,E1 -422.796,E2 -422.796} C_VEL
LIN {X 0,Y 608.443,Z 193.693,A -85,B 0,C 180,E1 -425.428,E2 -425.428} C_VEL
LIN {X 0,Y 608.459,Z 193.815,A -85,B 0,C 180,E1 -426.921,E2 -426.921} C_VEL
LIN {X 0,Y 608.584,Z 209.438,A -85,B 0,C 180,E1 -429.022,E2 -429.022} C_VEL
LIN {X 0,Y 608.522,Z 230.711,A -85,B 0,C 180,E1 -431.83,E2 -431.83} C_VEL
LIN {X 0,Y 608.491,Z 251.985,A -85,B 0,C 180,E1 -434.594,E2 -434.594} C_VEL
LIN {X 0,Y 608.45,Z 270.516,A -85,B 0,C 180,E1 -436.972,E2 -436.972} C_VEL
LIN {X 0,Y 608.543,Z 378.909,A -85,B 0,C 180,E1 -438.276,E2 -438.276} C_VEL
LIN {X 0,Y 608.509,Z 392.19,A -85,B 0,C 180,E1 -438.571,E2 -438.571} C_VEL
LIN {X 0,Y 608.514,Z 404.627,A -85,B 0,C 180,E1 -438.982,E2 -438.982} C_VEL
LIN {X 0,Y 608.5,Z 416.621,A -85,B 0,C 180,E1 -439.518,E2 -439.518} C_VEL
LIN {X 0,Y 608.488,Z 428.187,A -85,B 0,C 180,E1 -440.19,E2 -440.19} C_VEL
LIN {X 0,Y 608.485,Z 438.585,A -85,B 0,C 180,E1 -440.945,E2 -440.945} C_VEL
LIN {X 0,Y 608.475,Z 447.104,A -85,B 0,C 180,E1 -441.698,E2 -441.698} C_VEL
LIN {X 0,Y 608.471,Z 454.954,A -85,B 0,C 180,E1 -442.533,E2 -442.533} C_VEL
LIN {X 0,Y 608.461,Z 462.284,A -85,B 0,C 180,E1 -443.484,E2 -443.484} C_VEL
LIN {X 0,Y 608.451,Z 467.862,A -85,B 0,C 180,E1 -444.365,E2 -444.365} C_VEL
LIN {X 0,Y 608.432,Z 472.947,A -85,B 0,C 180,E1 -445.361,E2 -445.361} C_VEL
LIN {X 0,Y 608.449,Z 476.894,A -85,B 0,C 180,E1 -446.357,E2 -446.357} C_VEL
LIN {X 0,Y 608.425,Z 479.807,A -85,B 0,C 180,E1 -447.351,E2 -447.351} C_VEL
LIN {X 0,Y 608.445,Z 481.2,A -85,B 0,C 180,E1 -448.013,E2 -448.013} C_VEL
LIN {X 0,Y 608.439,Z 482.783,A -85,B 0,C 180,E1 -449.337,E2 -449.337} C_VEL
LIN {X 0,Y 608.434,Z 483,A -85,B 0,C 180,E1 -449.999,E2 -449.999} C_VEL
LIN {X 0,Y 608.448,Z 482.185,A -85,B 0,C 180,E1 -451.323,E2 -451.323} C_VEL
LIN {X 0,Y 608.444,Z 481.203,A -85,B 0,C 180,E1 -451.985,E2 -451.985} C_VEL
LIN {X 0,Y 608.425,Z 479.811,A -85,B 0,C 180,E1 -452.648,E2 -452.648} C_VEL
LIN {X 0,Y 608.449,Z 476.899,A -85,B 0,C 180,E1 -453.642,E2 -453.642} C_VEL
LIN {X 0,Y 608.432,Z 472.953,A -85,B 0,C 180,E1 -454.637,E2 -454.637} C_VEL
LIN {X 0,Y 608.438,Z 466.881,A -85,B 0,C 180,E1 -455.8,E2 -455.8} C_VEL
LIN {X 0,Y 608.461,Z 460.241,A -85,B 0,C 180,E1 -456.799,E2 -456.799} C_VEL
LIN {X 0,Y 608.455,Z 451.996,A -85,B 0,C 180,E1 -457.799,E2 -457.799} C_VEL
LIN {X 0,Y 608.472,Z 443.545,A -85,B 0,C 180,E1 -458.635,E2 -458.635} C_VEL
LIN {X 0,Y 608.479,Z 433.102,A -85,B 0,C 180,E1 -459.473,E2 -459.473} C_VEL
LIN {X 0,Y 608.492,Z 422.769,A -85,B 0,C 180,E1 -460.144,E2 -460.144} C_VEL
LIN {X 0,Y 608.519,Z 411.282,A -85,B 0,C 180,E1 -460.739,E2 -460.739} C_VEL
LIN {X 0,Y 608.526,Z 398.912,A -85,B 0,C 180,E1 -461.224,E2 -461.224} C_VEL
LIN {X 0,Y 608.54,Z 385.474,A -85,B 0,C 180,E1 -461.596,E2 -461.596} C_VEL
LIN {X 0,Y 608.55,Z 373.145,A -85,B 0,C 180,E1 -461.807,E2 -461.807} C_VEL
LIN {X 0,Y 608.438,Z 270.445,A -85,B 0,C 180,E1 -463.038,E2 -463.038} C_VEL
LIN {X 0,Y 608.504,Z 249.337,A -85,B 0,C 180,E1 -465.748,E2 -465.748} C_VEL
LIN {X 0,Y 608.5,Z 228.264,A -85,B 0,C 180,E1 -468.492,E2 -468.492} C_VEL
LIN {X 0,Y 608.562,Z 208.12,A -85,B 0,C 180,E1 -471.154,E2 -471.154} C_VEL
LIN {X 0,Y 608.456,Z 193.744,A -85,B 0,C 180,E1 -473.089,E2 -473.089} C_VEL
LIN {X 0,Y 608.478,Z 193.689,A -85,B 0,C 180,E1 -475.722,E2 -475.722} C_VEL
LIN {X 0,Y 608.449,Z 193.69,A -85,B 0,C 180,E1 -478.615,E2 -478.615} C_VEL
LIN {X 0,Y 608.441,Z 193.69,A -85,B 0,C 180,E1 -481.317,E2 -481.317} C_VEL
LIN {X 0,Y 608.477,Z 193.692,A -85,B 0,C 180,E1 -483.735,E2 -483.735} C_VEL
LIN {X 0,Y 608.438,Z 193.695,A -85,B 0,C 180,E1 -486.092,E2 -486.092} C_VEL
LIN {X 0,Y 608.415,Z 193.692,A -85,B 0,C 180,E1 -488.591,E2 -488.591} C_VEL
LIN {X 0,Y 608.46,Z 193.691,A -85,B 0,C 180,E1 -491.342,E2 -491.342} C_VEL
LIN {X 0,Y 608.448,Z 193.694,A -85,B 0,C 180,E1 -493.87,E2 -493.87} C_VEL
LIN {X 0,Y 608.44,Z 193.689,A -85,B 0,C 180,E1 -496.693,E2 -496.693} C_VEL
LIN {X 0,Y 608.446,Z 193.694,A -85,B 0,C 180,E1 -499.696,E2 -499.696} C_VEL
LIN {X 0,Y 608.428,Z 193.691,A -85,B 0,C 180,E1 -502.251,E2 -502.251} C_VEL
LIN {X 0,Y 608.454,Z 193.694,A -85,B 0,C 180,E1 -505.092,E2 -505.092} C_VEL
LIN {X 0,Y 608.423,Z 193.692,A -85,B 0,C 180,E1 -507.903,E2 -507.903} C_VEL
LIN {X 0,Y 608.411,Z 193.693,A -85,B 0,C 180,E1 -510.217,E2 -510.217} C_VEL
LIN {X 0,Y 608.455,Z 193.693,A -85,B 0,C 180,E1 -512.795,E2 -512.795} C_VEL
LIN {X 0,Y 608.423,Z 193.694,A -85,B 0,C 180,E1 -515.428,E2 -515.428} C_VEL
LIN {X 0,Y 608.423,Z 193.693,A -85,B 0,C 180,E1 -518.307,E2 -518.307} C_VEL
LIN {X 0,Y 608.411,Z 193.696,A -85,B 0,C 180,E1 -521.298,E2 -521.298} C_VEL
LIN {X 0,Y 608.4,Z 193.694,A -85,B 0,C 180,E1 -523.905,E2 -523.905} C_VEL
LIN {X 0,Y 608.452,Z 193.698,A -85,B 0,C 180,E1 -526.643,E2 -526.643} C_VEL
LIN {X 0,Y 608.41,Z 193.693,A -85,B 0,C 180,E1 -529.349,E2 -529.349} C_VEL
LIN {X 0,Y 608.406,Z 193.694,A -85,B 0,C 180,E1 -531.363,E2 -531.363} C_VEL
LIN {X 0,Y 608.425,Z 193.695,A -85,B 0,C 180,E1 -534.033,E2 -534.033} C_VEL
LIN {X 0,Y 608.466,Z 193.691,A -85,B 0,C 180,E1 -536.689,E2 -536.689} C_VEL
LIN {X 0,Y 608.408,Z 193.693,A -85,B 0,C 180,E1 -539.338,E2 -539.338} C_VEL
LIN {X 0,Y 608.421,Z 193.691,A -85,B 0,C 180,E1 -541.324,E2 -541.324} C_VEL
LIN {X 0,Y 608.439,Z 193.696,A -85,B 0,C 180,E1 -543.974,E2 -543.974} C_VEL
LIN {X 0,Y 608.451,Z 193.69,A -85,B 0,C 180,E1 -546.633,E2 -546.633} C_VEL
LIN {X 0,Y 608.432,Z 193.691,A -85,B 0,C 180,E1 -549.307,E2 -549.307} C_VEL
LIN {X 0,Y 608.429,Z 193.693,A -85,B 0,C 180,E1 -549.457,E2 -549.457} C_VEL
LIN {X 0,Y 607.77,Z 193.783,A -85,B 0,C 180,E1 -550.01,E2 -550.01} C_VEL
LIN {X 0,Y 604.929,Z 194.138,A -85,B 0,C 180,E1 -550.907,E2 -550.907} C_VEL
LIN {X 0,Y 602.523,Z 194.436,A -85,B 0,C 180,E1 -551.628,E2 -551.628} C_VEL
LIN {X 0,Y 601.484,Z 194.562,A -85,B 0,C 180,E1 -552.185,E2 -552.185} C_VEL
LIN {X 0,Y 601.396,Z 194.57,A -85,B 0,C 180,E1 -552.373,E2 -552.373} C_VEL
LIN {X 0,Y 601.409,Z 194.565,A -85,B 0,C 180,E1 -554.898,E2 -554.898} C_VEL
LIN {X 0,Y 601.398,Z 194.566,A -85,B 0,C 180,E1 -556.987,E2 -556.987} C_VEL
LIN {X 0,Y 601.396,Z 194.575,A -85,B 0,C 180,E1 -559.81,E2 -559.81} C_VEL
LIN {X 0,Y 601.403,Z 194.566,A -85,B 0,C 180,E1 -562.684,E2 -562.684} C_VEL
LIN {X 0,Y 601.39,Z 194.568,A -85,B 0,C 180,E1 -564.879,E2 -564.879} C_VEL
LIN {X 0,Y 601.406,Z 194.574,A -85,B 0,C 180,E1 -567.363,E2 -567.363} C_VEL
LIN {X 0,Y 601.423,Z 194.564,A -85,B 0,C 180,E1 -570.165,E2 -570.165} C_VEL
LIN {X 0,Y 601.406,Z 194.567,A -85,B 0,C 180,E1 -572.715,E2 -572.715} C_VEL
LIN {X 0,Y 601.387,Z 194.575,A -85,B 0,C 180,E1 -575.112,E2 -575.112} C_VEL
LIN {X 0,Y 601.432,Z 194.568,A -85,B 0,C 180,E1 -577.42,E2 -577.42} C_VEL
LIN {X 0,Y 601.409,Z 194.565,A -85,B 0,C 180,E1 -579.996,E2 -579.996} C_VEL
LIN {X 0,Y 601.405,Z 194.57,A -85,B 0,C 180,E1 -582.671,E2 -582.671} C_VEL
LIN {X 0,Y 601.423,Z 194.566,A -85,B 0,C 180,E1 -585.483,E2 -585.483} C_VEL
LIN {X 0,Y 601.42,Z 194.567,A -85,B 0,C 180,E1 -588.408,E2 -588.408} C_VEL
LIN {X 0,Y 601.43,Z 194.563,A -85,B 0,C 180,E1 -591.53,E2 -591.53} C_VEL
LIN {X 0,Y 601.385,Z 194.571,A -85,B 0,C 180,E1 -594.246,E2 -594.246} C_VEL
LIN {X 0,Y 601.42,Z 194.574,A -85,B 0,C 180,E1 -596.687,E2 -596.687} C_VEL
LIN {X 0,Y 601.439,Z 194.751,A -85,B 0,C 180,E1 -597.931,E2 -597.931} C_VEL
LIN {X 0,Y 601.443,Z 208.665,A -85,B 0,C 180,E1 -600.419,E2 -600.419} C_VEL
LIN {X 0,Y 601.405,Z 222.64,A -85,B 0,C 180,E1 -602.888,E2 -602.888} C_VEL
LIN {X 0,Y 601.651,Z 228.774,A -85,B 0,C 180,E1 -602.97,E2 -602.97} C_VEL
LIN {X 0,Y 601.544,Z 328.743,A -85,B 0,C 180,E1 -604.18,E2 -604.18} C_VEL
LIN {X 0,Y 601.514,Z 342.174,A -85,B 0,C 180,E1 -604.48,E2 -604.48} C_VEL
LIN {X 0,Y 601.532,Z 354.631,A -85,B 0,C 180,E1 -604.897,E2 -604.897} C_VEL
LIN {X 0,Y 601.485,Z 366.927,A -85,B 0,C 180,E1 -605.456,E2 -605.456} C_VEL
LIN {X 0,Y 601.451,Z 378.428,A -85,B 0,C 180,E1 -606.135,E2 -606.135} C_VEL
LIN {X 0,Y 601.44,Z 389.484,A -85,B 0,C 180,E1 -606.956,E2 -606.956} C_VEL
LIN {X 0,Y 601.415,Z 399.257,A -85,B 0,C 180,E1 -607.863,E2 -607.863} C_VEL
LIN {X 0,Y 601.387,Z 408.211,A -85,B 0,C 180,E1 -608.893,E2 -608.893} C_VEL
LIN {X 0,Y 601.369,Z 415.897,A -85,B 0,C 180,E1 -610.012,E2 -610.012} C_VEL
LIN {X 0,Y 601.347,Z 422.261,A -85,B 0,C 180,E1 -611.202,E2 -611.202} C_VEL
LIN {X 0,Y 601.328,Z 426.728,A -85,B 0,C 180,E1 -612.31,E2 -612.31} C_VEL
LIN {X 0,Y 601.325,Z 429.922,A -85,B 0,C 180,E1 -613.413,E2 -613.413} C_VEL
LIN {X 0,Y 601.326,Z 431.811,A -85,B 0,C 180,E1 -614.407,E2 -614.407} C_VEL
LIN {X 0,Y 601.315,Z 432.593,A -85,B 0,C 180,E1 -615.101,E2 -615.101} C_VEL
LIN {X 0,Y 601.352,Z 432.981,A -85,B 0,C 180,E1 -615.937,E2 -615.937} C_VEL
LIN {X 0,Y 601.325,Z 432.432,A -85,B 0,C 180,E1 -617.171,E2 -617.171} C_VEL
LIN {X 0,Y 601.342,Z 431.525,A -85,B 0,C 180,E1 -617.857,E2 -617.857} C_VEL
LIN {X 0,Y 601.336,Z 428.993,A -85,B 0,C 180,E1 -619.035,E2 -619.035} C_VEL
LIN {X 0,Y 601.342,Z 425.02,A -85,B 0,C 180,E1 -620.244,E2 -620.244} C_VEL
LIN {X 0,Y 601.382,Z 420.456,A -85,B 0,C 180,E1 -621.262,E2 -621.262} C_VEL
LIN {X 0,Y 601.38,Z 413.563,A -85,B 0,C 180,E1 -622.446,E2 -622.446} C_VEL
LIN {X 0,Y 601.378,Z 406.631,A -85,B 0,C 180,E1 -623.394,E2 -623.394} C_VEL
LIN {X 0,Y 601.428,Z 398.548,A -85,B 0,C 180,E1 -624.3,E2 -624.3} C_VEL
LIN {X 0,Y 601.442,Z 389.401,A -85,B 0,C 180,E1 -625.141,E2 -625.141} C_VEL
LIN {X 0,Y 601.443,Z 378.046,A -85,B 0,C 180,E1 -625.98,E2 -625.98} C_VEL
LIN {X 0,Y 601.487,Z 366.594,A -85,B 0,C 180,E1 -626.652,E2 -626.652} C_VEL
LIN {X 0,Y 601.551,Z 354.52,A -85,B 0,C 180,E1 -627.197,E2 -627.197} C_VEL
LIN {X 0,Y 601.541,Z 341.223,A -85,B 0,C 180,E1 -627.636,E2 -627.636} C_VEL
LIN {X 0,Y 601.589,Z 328.782,A -85,B 0,C 180,E1 -627.909,E2 -627.909} C_VEL
LIN {X 0,Y 601.549,Z 223.554,A -85,B 0,C 180,E1 -629.185,E2 -629.185} C_VEL
LIN {X 0,Y 601.408,Z 222.622,A -85,B 0,C 180,E1 -629.206,E2 -629.206} C_VEL
LIN {X 0,Y 601.436,Z 206.759,A -85,B 0,C 180,E1 -632.01,E2 -632.01} C_VEL
LIN {X 0,Y 601.414,Z 194.567,A -85,B 0,C 180,E1 -634.21,E2 -634.21} C_VEL
LIN {X 0,Y 601.409,Z 194.566,A -85,B 0,C 180,E1 -636.712,E2 -636.712} C_VEL
LIN {X 0,Y 601.415,Z 194.574,A -85,B 0,C 180,E1 -639.417,E2 -639.417} C_VEL
LIN {X 0,Y 601.4,Z 194.567,A -85,B 0,C 180,E1 -642.144,E2 -642.144} C_VEL
LIN {X 0,Y 601.406,Z 194.571,A -85,B 0,C 180,E1 -644.898,E2 -644.898} C_VEL
LIN {X 0,Y 601.414,Z 194.573,A -85,B 0,C 180,E1 -646.987,E2 -646.987} C_VEL
LIN {X 0,Y 601.386,Z 194.569,A -85,B 0,C 180,E1 -649.811,E2 -649.811} C_VEL
LIN {X 0,Y 601.383,Z 194.568,A -85,B 0,C 180,E1 -651.961,E2 -651.961} C_VEL
LIN {X 0,Y 601.388,Z 194.578,A -85,B 0,C 180,E1 -654.88,E2 -654.88} C_VEL
LIN {X 0,Y 601.385,Z 194.571,A -85,B 0,C 180,E1 -657.356,E2 -657.356} C_VEL
LIN {X 0,Y 601.377,Z 194.571,A -85,B 0,C 180,E1 -659.396,E2 -659.396} C_VEL
LIN {X 0,Y 601.391,Z 194.568,A -85,B 0,C 180,E1 -661.728,E2 -661.728} C_VEL
LIN {X 0,Y 601.388,Z 194.57,A -85,B 0,C 180,E1 -664.122,E2 -664.122} C_VEL
LIN {X 0,Y 601.386,Z 194.578,A -85,B 0,C 180,E1 -666.585,E2 -666.585} C_VEL
LIN {X 0,Y 601.377,Z 194.571,A -85,B 0,C 180,E1 -669.13,E2 -669.13} C_VEL
LIN {X 0,Y 601.389,Z 194.569,A -85,B 0,C 180,E1 -671.769,E2 -671.769} C_VEL
LIN {X 0,Y 601.405,Z 194.573,A -85,B 0,C 180,E1 -674.533,E2 -674.533} C_VEL
LIN {X 0,Y 601.345,Z 194.573,A -85,B 0,C 180,E1 -677.323,E2 -677.323} C_VEL
LIN {X 0,Y 601.379,Z 194.576,A -85,B 0,C 180,E1 -680.002,E2 -680.002} C_VEL
LIN {X 0,Y 601.364,Z 194.573,A -85,B 0,C 180,E1 -682.628,E2 -682.628} C_VEL
LIN {X 0,Y 601.353,Z 194.572,A -85,B 0,C 180,E1 -685.064,E2 -685.064} C_VEL
LIN {X 0,Y 601.396,Z 194.57,A -85,B 0,C 180,E1 -687.482,E2 -687.482} C_VEL
LIN {X 0,Y 601.409,Z 194.575,A -85,B 0,C 180,E1 -689.856,E2 -689.856} C_VEL
LIN {X 0,Y 601.371,Z 194.57,A -85,B 0,C 180,E1 -692.885,E2 -692.885} C_VEL
LIN {X 0,Y 601.458,Z 194.568,A -85,B 0,C 180,E1 -695.859,E2 -695.859} C_VEL
LIN {X 0,Y 601.383,Z 194.569,A -85,B 0,C 180,E1 -698.76,E2 -698.76} C_VEL
LIN {X 0,Y 601.401,Z 194.585,A -85,B 0,C 180,E1 -700.9,E2 -700.9} C_VEL
LIN {X 0,Y 601.452,Z 210.318,A -85,B 0,C 180,E1 -703.713,E2 -703.713} C_VEL
LIN {X 0,Y 601.461,Z 222.904,A -85,B 0,C 180,E1 -705.895,E2 -705.895} C_VEL
LIN {X 0,Y 601.666,Z 242.569,A -85,B 0,C 180,E1 -706.136,E2 -706.136} C_VEL
LIN {X 0,Y 601.594,Z 329.65,A -85,B 0,C 180,E1 -707.197,E2 -707.197} C_VEL
LIN {X 0,Y 601.58,Z 343.485,A -85,B 0,C 180,E1 -707.518,E2 -707.518} C_VEL
LIN {X 0,Y 601.563,Z 355.829,A -85,B 0,C 180,E1 -707.946,E2 -707.946} C_VEL
LIN {X 0,Y 601.502,Z 366.956,A -85,B 0,C 180,E1 -708.458,E2 -708.458} C_VEL
LIN {X 0,Y 601.458,Z 378.401,A -85,B 0,C 180,E1 -709.134,E2 -709.134} C_VEL
LIN {X 0,Y 601.44,Z 388.849,A -85,B 0,C 180,E1 -709.905,E2 -709.905} C_VEL
LIN {X 0,Y 601.413,Z 398.2,A -85,B 0,C 180,E1 -710.753,E2 -710.753} C_VEL
LIN {X 0,Y 601.403,Z 407.222,A -85,B 0,C 180,E1 -711.769,E2 -711.769} C_VEL
LIN {X 0,Y 601.389,Z 414.483,A -85,B 0,C 180,E1 -712.783,E2 -712.783} C_VEL
LIN {X 0,Y 601.361,Z 419.28,A -85,B 0,C 180,E1 -713.606,E2 -713.606} C_VEL
LIN {X 0,Y 601.355,Z 424.144,A -85,B 0,C 180,E1 -714.635,E2 -714.635} C_VEL
LIN {X 0,Y 601.356,Z 427.786,A -85,B 0,C 180,E1 -715.643,E2 -715.643} C_VEL
LIN {X 0,Y 601.34,Z 430.426,A -85,B 0,C 180,E1 -716.65,E2 -716.65} C_VEL
LIN {X 0,Y 601.324,Z 431.671,A -85,B 0,C 180,E1 -717.32,E2 -717.32} C_VEL
LIN {X 0,Y 601.34,Z 432.509,A -85,B 0,C 180,E1 -717.991,E2 -717.991} C_VEL
LIN {X 0,Y 601.339,Z 432.94,A -85,B 0,C 180,E1 -719.33,E2 -719.33} C_VEL
LIN {X 0,Y 601.336,Z 432.587,A -85,B 0,C 180,E1 -720,E2 -720} C_VEL
LIN {X 0,Y 601.339,Z 431.83,A -85,B 0,C 180,E1 -720.669,E2 -720.669} C_VEL
LIN {X 0,Y 601.345,Z 429.063,A -85,B 0,C 180,E1 -722.009,E2 -722.009} C_VEL
LIN {X 0,Y 601.379,Z 425.869,A -85,B 0,C 180,E1 -723.014,E2 -723.014} C_VEL
LIN {X 0,Y 601.346,Z 421.619,A -85,B 0,C 180,E1 -724.021,E2 -724.021} C_VEL
LIN {X 0,Y 601.361,Z 415.173,A -85,B 0,C 180,E1 -725.196,E2 -725.196} C_VEL
LIN {X 0,Y 601.378,Z 408.043,A -85,B 0,C 180,E1 -726.219,E2 -726.219} C_VEL
LIN {X 0,Y 601.418,Z 399.357,A -85,B 0,C 180,E1 -727.217,E2 -727.217} C_VEL
LIN {X 0,Y 601.453,Z 390.355,A -85,B 0,C 180,E1 -728.06,E2 -728.06} C_VEL
LIN {X 0,Y 601.447,Z 380.404,A -85,B 0,C 180,E1 -728.822,E2 -728.822} C_VEL
LIN {X 0,Y 601.492,Z 369.408,A -85,B 0,C 180,E1 -729.499,E2 -729.499} C_VEL
LIN {X 0,Y 601.519,Z 357.091,A -85,B 0,C 180,E1 -730.093,E2 -730.093} C_VEL
LIN {X 0,Y 601.558,Z 345.299,A -85,B 0,C 180,E1 -730.518,E2 -730.518} C_VEL
LIN {X 0,Y 601.547,Z 332.607,A -85,B 0,C 180,E1 -730.839,E2 -730.839} C_VEL
LIN {X 0,Y 601.593,Z 314.741,A -85,B 0,C 180,E1 -731.091,E2 -731.091} C_VEL
LIN {X 0,Y 601.51,Z 223.761,A -85,B 0,C 180,E1 -732.183,E2 -732.183} C_VEL
LIN {X 0,Y 601.351,Z 222.494,A -85,B 0,C 180,E1 -732.229,E2 -732.229} C_VEL
LIN {X 0,Y 601.447,Z 207.394,A -85,B 0,C 180,E1 -734.896,E2 -734.896} C_VEL
LIN {X 0,Y 601.458,Z 194.561,A -85,B 0,C 180,E1 -737.204,E2 -737.204} C_VEL
LIN {X 0,Y 601.4,Z 194.568,A -85,B 0,C 180,E1 -739.81,E2 -739.81} C_VEL
LIN {X 0,Y 601.421,Z 194.571,A -85,B 0,C 180,E1 -742.605,E2 -742.605} C_VEL
LIN {X 0,Y 601.402,Z 194.569,A -85,B 0,C 180,E1 -744.879,E2 -744.879} C_VEL
LIN {X 0,Y 601.416,Z 194.564,A -85,B 0,C 180,E1 -747.361,E2 -747.361} C_VEL
LIN {X 0,Y 601.409,Z 194.565,A -85,B 0,C 180,E1 -749.394,E2 -749.394} C_VEL
LIN {X 0,Y 601.402,Z 194.568,A -85,B 0,C 180,E1 -751.727,E2 -751.727} C_VEL
LIN {X 0,Y 601.424,Z 194.571,A -85,B 0,C 180,E1 -754.119,E2 -754.119} C_VEL
LIN {X 0,Y 601.436,Z 194.562,A -85,B 0,C 180,E1 -757.381,E2 -757.381} C_VEL
LIN {X 0,Y 601.402,Z 194.573,A -85,B 0,C 180,E1 -759.996,E2 -759.996} C_VEL
LIN {X 0,Y 601.412,Z 194.567,A -85,B 0,C 180,E1 -762.67,E2 -762.67} C_VEL
LIN {X 0,Y 601.403,Z 194.567,A -85,B 0,C 180,E1 -765.479,E2 -765.479} C_VEL
LIN {X 0,Y 601.425,Z 194.568,A -85,B 0,C 180,E1 -768.407,E2 -768.407} C_VEL
LIN {X 0,Y 601.403,Z 194.566,A -85,B 0,C 180,E1 -770.872,E2 -770.872} C_VEL
LIN {X 0,Y 601.393,Z 194.569,A -85,B 0,C 180,E1 -773.416,E2 -773.416} C_VEL
LIN {X 0,Y 601.437,Z 194.57,A -85,B 0,C 180,E1 -776.064,E2 -776.064} C_VEL
LIN {X 0,Y 601.411,Z 194.566,A -85,B 0,C 180,E1 -779.057,E2 -779.057} C_VEL
LIN {X 0,Y 601.415,Z 194.568,A -85,B 0,C 180,E1 -781.372,E2 -781.372} C_VEL
LIN {X 0,Y 601.437,Z 194.564,A -85,B 0,C 180,E1 -784.382,E2 -784.382} C_VEL
LIN {X 0,Y 601.415,Z 194.646,A -85,B 0,C 180,E1 -786.748,E2 -786.748} C_VEL
LIN {X 0,Y 601.691,Z 199.714,A -85,B 0,C 180,E1 -787.452,E2 -787.452} C_VEL
LIN {X 0,Y 601.595,Z 218.745,A -85,B 0,C 180,E1 -790.018,E2 -790.018} C_VEL
LIN {X 0,Y 601.537,Z 238.689,A -85,B 0,C 180,E1 -792.666,E2 -792.666} C_VEL
LIN {X 0,Y 601.471,Z 258.633,A -85,B 0,C 180,E1 -795.277,E2 -795.277} C_VEL
LIN {X 0,Y 601.414,Z 270.433,A -85,B 0,C 180,E1 -796.806,E2 -796.806} C_VEL
LIN {X 0,Y 601.642,Z 276.45,A -85,B 0,C 180,E1 -796.897,E2 -796.897} C_VEL
LIN {X 0,Y 601.613,Z 378.908,A -85,B 0,C 180,E1 -798.139,E2 -798.139} C_VEL
LIN {X 0,Y 601.572,Z 392.19,A -85,B 0,C 180,E1 -798.437,E2 -798.437} C_VEL
LIN {X 0,Y 601.543,Z 404.625,A -85,B 0,C 180,E1 -798.853,E2 -798.853} C_VEL
LIN {X 0,Y 601.523,Z 416.62,A -85,B 0,C 180,E1 -799.395,E2 -799.395} C_VEL
LIN {X 0,Y 601.487,Z 428.188,A -85,B 0,C 180,E1 -800.075,E2 -800.075} C_VEL
LIN {X 0,Y 601.445,Z 438.586,A -85,B 0,C 180,E1 -800.838,E2 -800.838} C_VEL
LIN {X 0,Y 601.429,Z 447.105,A -85,B 0,C 180,E1 -801.6,E2 -801.6} C_VEL
LIN {X 0,Y 601.418,Z 454.954,A -85,B 0,C 180,E1 -802.445,E2 -802.445} C_VEL
LIN {X 0,Y 601.37,Z 462.221,A -85,B 0,C 180,E1 -803.397,E2 -803.397} C_VEL
LIN {X 0,Y 601.372,Z 467.862,A -85,B 0,C 180,E1 -804.298,E2 -804.298} C_VEL
LIN {X 0,Y 601.336,Z 472.947,A -85,B 0,C 180,E1 -805.307,E2 -805.307} C_VEL
LIN {X 0,Y 601.368,Z 476.894,A -85,B 0,C 180,E1 -806.314,E2 -806.314} C_VEL
LIN {X 0,Y 601.325,Z 479.808,A -85,B 0,C 180,E1 -807.32,E2 -807.32} C_VEL
LIN {X 0,Y 601.343,Z 481.201,A -85,B 0,C 180,E1 -807.99,E2 -807.99} C_VEL
LIN {X 0,Y 601.339,Z 482.783,A -85,B 0,C 180,E1 -809.33,E2 -809.33} C_VEL
LIN {X 0,Y 601.335,Z 483,A -85,B 0,C 180,E1 -809.999,E2 -809.999} C_VEL
LIN {X 0,Y 601.347,Z 482.185,A -85,B 0,C 180,E1 -811.339,E2 -811.339} C_VEL
LIN {X 0,Y 601.343,Z 481.203,A -85,B 0,C 180,E1 -812.009,E2 -812.009} C_VEL
LIN {X 0,Y 601.325,Z 479.811,A -85,B 0,C 180,E1 -812.679,E2 -812.679} C_VEL
LIN {X 0,Y 601.368,Z 476.898,A -85,B 0,C 180,E1 -813.685,E2 -813.685} C_VEL
LIN {X 0,Y 601.336,Z 472.953,A -85,B 0,C 180,E1 -814.692,E2 -814.692} C_VEL
LIN {X 0,Y 601.372,Z 466.882,A -85,B 0,C 180,E1 -815.868,E2 -815.868} C_VEL
LIN {X 0,Y 601.387,Z 460.241,A -85,B 0,C 180,E1 -816.879,E2 -816.879} C_VEL
LIN {X 0,Y 601.4,Z 451.996,A -85,B 0,C 180,E1 -817.892,E2 -817.892} C_VEL
LIN {X 0,Y 601.436,Z 443.546,A -85,B 0,C 180,E1 -818.737,E2 -818.737} C_VEL
LIN {X 0,Y 601.45,Z 433.104,A -85,B 0,C 180,E1 -819.584,E2 -819.584} C_VEL
LIN {X 0,Y 601.47,Z 422.771,A -85,B 0,C 180,E1 -820.264,E2 -820.264} C_VEL
LIN {X 0,Y 601.537,Z 410.607,A -85,B 0,C 180,E1 -820.896,E2 -820.896} C_VEL
LIN {X 0,Y 601.552,Z 398.242,A -85,B 0,C 180,E1 -821.378,E2 -821.378} C_VEL
LIN {X 0,Y 601.579,Z 385.474,A -85,B 0,C 180,E1 -821.732,E2 -821.732} C_VEL
LIN {X 0,Y 601.617,Z 373.145,A -85,B 0,C 180,E1 -821.945,E2 -821.945} C_VEL
LIN {X 0,Y 601.504,Z 271.21,A -85,B 0,C 180,E1 -823.169,E2 -823.169} C_VEL
LIN {X 0,Y 601.444,Z 270.279,A -85,B 0,C 180,E1 -823.213,E2 -823.213} C_VEL
LIN {X 0,Y 601.518,Z 248.008,A -85,B 0,C 180,E1 -826.11,E2 -826.11} C_VEL
LIN {X 0,Y 601.54,Z 227.219,A -85,B 0,C 180,E1 -828.852,E2 -828.852} C_VEL
LIN {X 0,Y 601.672,Z 206.79,A -85,B 0,C 180,E1 -831.588,E2 -831.588} C_VEL
LIN {X 0,Y 601.665,Z 196.153,A -85,B 0,C 180,E1 -833.035,E2 -833.035} C_VEL
LIN {X 0,Y 601.402,Z 194.57,A -85,B 0,C 180,E1 -833.273,E2 -833.273} C_VEL
LIN {X 0,Y 601.414,Z 194.571,A -85,B 0,C 180,E1 -835.867,E2 -835.867} C_VEL
LIN {X 0,Y 601.412,Z 194.566,A -85,B 0,C 180,E1 -838.784,E2 -838.784} C_VEL
LIN {X 0,Y 601.415,Z 194.567,A -85,B 0,C 180,E1 -841.454,E2 -841.454} C_VEL
LIN {X 0,Y 601.419,Z 194.57,A -85,B 0,C 180,E1 -844.118,E2 -844.118} C_VEL
LIN {X 0,Y 601.383,Z 194.569,A -85,B 0,C 180,E1 -846.583,E2 -846.583} C_VEL
LIN {X 0,Y 601.412,Z 194.571,A -85,B 0,C 180,E1 -849.532,E2 -849.532} C_VEL
LIN {X 0,Y 601.409,Z 194.574,A -85,B 0,C 180,E1 -851.765,E2 -851.765} C_VEL
LIN {X 0,Y 601.392,Z 194.567,A -85,B 0,C 180,E1 -854.532,E2 -854.532} C_VEL
LIN {X 0,Y 601.403,Z 194.575,A -85,B 0,C 180,E1 -857.409,E2 -857.409} C_VEL
LIN {X 0,Y 601.388,Z 194.57,A -85,B 0,C 180,E1 -860.003,E2 -860.003} C_VEL
LIN {X 0,Y 601.422,Z 194.564,A -85,B 0,C 180,E1 -862.618,E2 -862.618} C_VEL
LIN {X 0,Y 601.402,Z 194.567,A -85,B 0,C 180,E1 -865.88,E2 -865.88} C_VEL
LIN {X 0,Y 601.403,Z 194.567,A -85,B 0,C 180,E1 -868.546,E2 -868.546} C_VEL
LIN {X 0,Y 601.404,Z 194.571,A -85,B 0,C 180,E1 -871.372,E2 -871.372} C_VEL
LIN {X 0,Y 601.371,Z 194.571,A -85,B 0,C 180,E1 -873.635,E2 -873.635} C_VEL
LIN {X 0,Y 601.378,Z 194.569,A -85,B 0,C 180,E1 -875.856,E2 -875.856} C_VEL
LIN {X 0,Y 601.36,Z 194.57,A -85,B 0,C 180,E1 -878.039,E2 -878.039} C_VEL
LIN {X 0,Y 601.367,Z 194.571,A -85,B 0,C 180,E1 -880.189,E2 -880.189} C_VEL
LIN {X 0,Y 601.391,Z 194.573,A -85,B 0,C 180,E1 -883.013,E2 -883.013} C_VEL
LIN {X 0,Y 601.363,Z 194.57,A -85,B 0,C 180,E1 -885.927,E2 -885.927} C_VEL
LIN {X 0,Y 601.393,Z 194.571,A -85,B 0,C 180,E1 -888.999,E2 -888.999} C_VEL
LIN {X 0,Y 601.375,Z 194.57,A -85,B 0,C 180,E1 -891.262,E2 -891.262} C_VEL
LIN {X 0,Y 601.374,Z 194.569,A -85,B 0,C 180,E1 -893.384,E2 -893.384} C_VEL
LIN {X 0,Y 601.375,Z 194.572,A -85,B 0,C 180,E1 -895.979,E2 -895.979} C_VEL
LIN {X 0,Y 601.413,Z 194.569,A -85,B 0,C 180,E1 -898.661,E2 -898.661} C_VEL
LIN {X 0,Y 601.376,Z 194.569,A -85,B 0,C 180,E1 -901.339,E2 -901.339} C_VEL
LIN {X 0,Y 601.36,Z 194.57,A -85,B 0,C 180,E1 -903.35,E2 -903.35} C_VEL
LIN {X 0,Y 601.399,Z 194.575,A -85,B 0,C 180,E1 -906.037,E2 -906.037} C_VEL
LIN {X 0,Y 601.397,Z 194.567,A -85,B 0,C 180,E1 -908.738,E2 -908.738} C_VEL
LIN {X 0,Y 601.398,Z 194.568,A -85,B 0,C 180,E1 -911.459,E2 -911.459} C_VEL
LIN {X 0,Y 601.396,Z 194.57,A -85,B 0,C 180,E1 -912.373,E2 -912.373} C_VEL
LIN {X 0,Y 600.723,Z 194.653,A -85,B 0,C 180,E1 -912.932,E2 -912.932} C_VEL
LIN {X 0,Y 597.869,Z 195.016,A -85,B 0,C 180,E1 -913.84,E2 -913.84} C_VEL
LIN {X 0,Y 595.463,Z 195.31,A -85,B 0,C 180,E1 -914.571,E2 -914.571} C_VEL
LIN {X 0,Y 594.429,Z 195.436,A -85,B 0,C 180,E1 -915.134,E2 -915.134} C_VEL
LIN {X 0,Y 594.344,Z 195.448,A -85,B 0,C 180,E1 -915.325,E2 -915.325} C_VEL
LIN {X 0,Y 594.343,Z 195.452,A -85,B 0,C 180,E1 -917.906,E2 -917.906} C_VEL
LIN {X 0,Y 594.384,Z 195.44,A -85,B 0,C 180,E1 -920.777,E2 -920.777} C_VEL
LIN {X 0,Y 594.385,Z 195.448,A -85,B 0,C 180,E1 -923.705,E2 -923.705} C_VEL
LIN {X 0,Y 594.371,Z 195.442,A -85,B 0,C 180,E1 -926.701,E2 -926.701} C_VEL
LIN {X 0,Y 594.37,Z 195.445,A -85,B 0,C 180,E1 -928.999,E2 -928.999} C_VEL
LIN {X 0,Y 594.385,Z 195.446,A -85,B 0,C 180,E1 -931.646,E2 -931.646} C_VEL
LIN {X 0,Y 594.371,Z 195.442,A -85,B 0,C 180,E1 -934.581,E2 -934.581} C_VEL
LIN {X 0,Y 594.381,Z 195.449,A -85,B 0,C 180,E1 -937.087,E2 -937.087} C_VEL
LIN {X 0,Y 594.375,Z 195.443,A -85,B 0,C 180,E1 -939.776,E2 -939.776} C_VEL
LIN {X 0,Y 594.362,Z 195.444,A -85,B 0,C 180,E1 -942.377,E2 -942.377} C_VEL
LIN {X 0,Y 594.361,Z 195.45,A -85,B 0,C 180,E1 -945.192,E2 -945.192} C_VEL
LIN {X 0,Y 594.38,Z 195.442,A -85,B 0,C 180,E1 -948.153,E2 -948.153} C_VEL
LIN {X 0,Y 594.378,Z 195.445,A -85,B 0,C 180,E1 -951.196,E2 -951.196} C_VEL
LIN {X 0,Y 594.35,Z 195.445,A -85,B 0,C 180,E1 -953.757,E2 -953.757} C_VEL
LIN {X 0,Y 594.376,Z 195.445,A -85,B 0,C 180,E1 -956.24,E2 -956.24} C_VEL
LIN {X 0,Y 594.442,Z 195.562,A -85,B 0,C 180,E1 -957.858,E2 -957.858} C_VEL
LIN {X 0,Y 594.401,Z 209.73,A -85,B 0,C 180,E1 -960.421,E2 -960.421} C_VEL
LIN {X 0,Y 594.336,Z 222.644,A -85,B 0,C 180,E1 -962.729,E2 -962.729} C_VEL
LIN {X 0,Y 594.743,Z 227.229,A -85,B 0,C 180,E1 -962.797,E2 -962.797} C_VEL
LIN {X 0,Y 594.614,Z 329.116,A -85,B 0,C 180,E1 -964.046,E2 -964.046} C_VEL
LIN {X 0,Y 594.554,Z 342.346,A -85,B 0,C 180,E1 -964.347,E2 -964.347} C_VEL
LIN {X 0,Y 594.567,Z 354.762,A -85,B 0,C 180,E1 -964.77,E2 -964.77} C_VEL
LIN {X 0,Y 594.523,Z 366.165,A -85,B 0,C 180,E1 -965.291,E2 -965.291} C_VEL
LIN {X 0,Y 594.423,Z 377.112,A -85,B 0,C 180,E1 -965.928,E2 -965.928} C_VEL
LIN {X 0,Y 594.421,Z 388.419,A -85,B 0,C 180,E1 -966.76,E2 -966.76} C_VEL
LIN {X 0,Y 594.371,Z 397.886,A -85,B 0,C 180,E1 -967.622,E2 -967.622} C_VEL
LIN {X 0,Y 594.342,Z 407.102,A -85,B 0,C 180,E1 -968.667,E2 -968.667} C_VEL
LIN {X 0,Y 594.302,Z 414.838,A -85,B 0,C 180,E1 -969.764,E2 -969.764} C_VEL
LIN {X 0,Y 594.248,Z 421.211,A -85,B 0,C 180,E1 -970.923,E2 -970.923} C_VEL
LIN {X 0,Y 594.241,Z 426.103,A -85,B 0,C 180,E1 -972.092,E2 -972.092} C_VEL
LIN {X 0,Y 594.24,Z 429.805,A -85,B 0,C 180,E1 -973.333,E2 -973.333} C_VEL
LIN {X 0,Y 594.225,Z 431.532,A -85,B 0,C 180,E1 -974.216,E2 -974.216} C_VEL
LIN {X 0,Y 594.211,Z 432.447,A -85,B 0,C 180,E1 -974.919,E2 -974.919} C_VEL
LIN {X 0,Y 594.263,Z 432.968,A -85,B 0,C 180,E1 -975.877,E2 -975.877} C_VEL
LIN {X 0,Y 594.244,Z 432.582,A -85,B 0,C 180,E1 -977.015,E2 -977.015} C_VEL
LIN {X 0,Y 594.239,Z 431.799,A -85,B 0,C 180,E1 -977.709,E2 -977.709} C_VEL
LIN {X 0,Y 594.251,Z 429.182,A -85,B 0,C 180,E1 -978.998,E2 -978.998} C_VEL
LIN {X 0,Y 594.258,Z 425.634,A -85,B 0,C 180,E1 -980.127,E2 -980.127} C_VEL
LIN {X 0,Y 594.294,Z 421.257,A -85,B 0,C 180,E1 -981.157,E2 -981.157} C_VEL
LIN {X 0,Y 594.299,Z 415.694,A -85,B 0,C 180,E1 -982.185,E2 -982.185} C_VEL
LIN {X 0,Y 594.319,Z 408.769,A -85,B 0,C 180,E1 -983.21,E2 -983.21} C_VEL
LIN {X 0,Y 594.344,Z 400.14,A -85,B 0,C 180,E1 -984.232,E2 -984.232} C_VEL
LIN {X 0,Y 594.417,Z 391.318,A -85,B 0,C 180,E1 -985.083,E2 -985.083} C_VEL
LIN {X 0,Y 594.436,Z 381.698,A -85,B 0,C 180,E1 -985.848,E2 -985.848} C_VEL
LIN {X 0,Y 594.493,Z 371.14,A -85,B 0,C 180,E1 -986.527,E2 -986.527} C_VEL
LIN {X 0,Y 594.552,Z 359.458,A -85,B 0,C 180,E1 -987.121,E2 -987.121} C_VEL
LIN {X 0,Y 594.573,Z 347.396,A -85,B 0,C 180,E1 -987.587,E2 -987.587} C_VEL
LIN {X 0,Y 594.622,Z 334.098,A -85,B 0,C 180,E1 -987.948,E2 -987.948} C_VEL
LIN {X 0,Y 594.655,Z 320.901,A -85,B 0,C 180,E1 -988.159,E2 -988.159} C_VEL
LIN {X 0,Y 594.721,Z 224.775,A -85,B 0,C 180,E1 -989.324,E2 -989.324} C_VEL
LIN {X 0,Y 594.351,Z 222.617,A -85,B 0,C 180,E1 -989.366,E2 -989.366} C_VEL
LIN {X 0,Y 594.407,Z 207.703,A -85,B 0,C 180,E1 -992.033,E2 -992.033} C_VEL
LIN {X 0,Y 594.387,Z 195.443,A -85,B 0,C 180,E1 -994.26,E2 -994.26} C_VEL
LIN {X 0,Y 594.385,Z 195.442,A -85,B 0,C 180,E1 -996.791,E2 -996.791} C_VEL
LIN {X 0,Y 594.36,Z 195.451,A -85,B 0,C 180,E1 -999.529,E2 -999.529} C_VEL
LIN {X 0,Y 594.379,Z 195.441,A -85,B 0,C 180,E1 -1002.289,E2 -1002.289} C_VEL
LIN {X 0,Y 594.356,Z 195.453,A -85,B 0,C 180,E1 -1005.079,E2 -1005.079} C_VEL
LIN {X 0,Y 594.377,Z 195.451,A -85,B 0,C 180,E1 -1007.194,E2 -1007.194} C_VEL
LIN {X 0,Y 594.362,Z 195.443,A -85,B 0,C 180,E1 -1010.055,E2 -1010.055} C_VEL
LIN {X 0,Y 594.354,Z 195.454,A -85,B 0,C 180,E1 -1012.968,E2 -1012.968} C_VEL
LIN {X 0,Y 594.329,Z 195.453,A -85,B 0,C 180,E1 -1015.196,E2 -1015.196} C_VEL
LIN {X 0,Y 594.35,Z 195.446,A -85,B 0,C 180,E1 -1017.519,E2 -1017.519} C_VEL
LIN {X 0,Y 594.349,Z 195.445,A -85,B 0,C 180,E1 -1019.778,E2 -1019.778} C_VEL
LIN {X 0,Y 594.365,Z 195.445,A -85,B 0,C 180,E1 -1022.148,E2 -1022.148} C_VEL
LIN {X 0,Y 594.359,Z 195.453,A -85,B 0,C 180,E1 -1024.582,E2 -1024.582} C_VEL
LIN {X 0,Y 594.354,Z 195.444,A -85,B 0,C 180,E1 -1027.603,E2 -1027.603} C_VEL
LIN {X 0,Y 594.342,Z 195.447,A -85,B 0,C 180,E1 -1029.77,E2 -1029.77} C_VEL
LIN {X 0,Y 594.346,Z 195.455,A -85,B 0,C 180,E1 -1032.378,E2 -1032.378} C_VEL
LIN {X 0,Y 594.319,Z 195.449,A -85,B 0,C 180,E1 -1035.196,E2 -1035.196} C_VEL
LIN {X 0,Y 594.362,Z 195.452,A -85,B 0,C 180,E1 -1038.155,E2 -1038.155} C_VEL
LIN {X 0,Y 594.323,Z 195.448,A -85,B 0,C 180,E1 -1041.19,E2 -1041.19} C_VEL
LIN {X 0,Y 594.339,Z 195.451,A -85,B 0,C 180,E1 -1043.754,E2 -1043.754} C_VEL
LIN {X 0,Y 594.343,Z 195.452,A -85,B 0,C 180,E1 -1046.236,E2 -1046.236} C_VEL
LIN {X 0,Y 594.326,Z 195.449,A -85,B 0,C 180,E1 -1048.647,E2 -1048.647} C_VEL
LIN {X 0,Y 594.338,Z 195.447,A -85,B 0,C 180,E1 -1051.051,E2 -1051.051} C_VEL
LIN {X 0,Y 594.337,Z 195.453,A -85,B 0,C 180,E1 -1053.988,E2 -1053.988} C_VEL
LIN {X 0,Y 594.364,Z 195.445,A -85,B 0,C 180,E1 -1056.295,E2 -1056.295} C_VEL
LIN {X 0,Y 594.394,Z 195.443,A -85,B 0,C 180,E1 -1059.224,E2 -1059.224} C_VEL
LIN {X 0,Y 594.345,Z 195.514,A -85,B 0,C 180,E1 -1060.847,E2 -1060.847} C_VEL
LIN {X 0,Y 594.429,Z 208.895,A -85,B 0,C 180,E1 -1063.272,E2 -1063.272} C_VEL
LIN {X 0,Y 594.373,Z 222.607,A -85,B 0,C 180,E1 -1065.723,E2 -1065.723} C_VEL
LIN {X 0,Y 594.768,Z 227.761,A -85,B 0,C 180,E1 -1065.804,E2 -1065.804} C_VEL
LIN {X 0,Y 594.664,Z 328.933,A -85,B 0,C 180,E1 -1067.045,E2 -1067.045} C_VEL
LIN {X 0,Y 594.64,Z 342.324,A -85,B 0,C 180,E1 -1067.348,E2 -1067.348} C_VEL
LIN {X 0,Y 594.588,Z 354.435,A -85,B 0,C 180,E1 -1067.759,E2 -1067.759} C_VEL
LIN {X 0,Y 594.514,Z 366.737,A -85,B 0,C 180,E1 -1068.32,E2 -1068.32} C_VEL
LIN {X 0,Y 594.427,Z 378.155,A -85,B 0,C 180,E1 -1068.999,E2 -1068.999} C_VEL
LIN {X 0,Y 594.413,Z 388.696,A -85,B 0,C 180,E1 -1069.784,E2 -1069.784} C_VEL
LIN {X 0,Y 594.366,Z 398.078,A -85,B 0,C 180,E1 -1070.643,E2 -1070.643} C_VEL
LIN {X 0,Y 594.327,Z 407.134,A -85,B 0,C 180,E1 -1071.671,E2 -1071.671} C_VEL
LIN {X 0,Y 594.3,Z 414.404,A -85,B 0,C 180,E1 -1072.696,E2 -1072.696} C_VEL
LIN {X 0,Y 594.267,Z 419.719,A -85,B 0,C 180,E1 -1073.623,E2 -1073.623} C_VEL
LIN {X 0,Y 594.276,Z 424.095,A -85,B 0,C 180,E1 -1074.571,E2 -1074.571} C_VEL
LIN {X 0,Y 594.271,Z 427.746,A -85,B 0,C 180,E1 -1075.591,E2 -1075.591} C_VEL
LIN {X 0,Y 594.26,Z 430.397,A -85,B 0,C 180,E1 -1076.61,E2 -1076.61} C_VEL
LIN {X 0,Y 594.224,Z 431.655,A -85,B 0,C 180,E1 -1077.288,E2 -1077.288} C_VEL
LIN {X 0,Y 594.238,Z 432.497,A -85,B 0,C 180,E1 -1077.967,E2 -1077.967} C_VEL
LIN {X 0,Y 594.249,Z 432.913,A -85,B 0,C 180,E1 -1078.644,E2 -1078.644} C_VEL
LIN {X 0,Y 594.237,Z 432.596,A -85,B 0,C 180,E1 -1080,E2 -1080} C_VEL
LIN {X 0,Y 594.24,Z 431.837,A -85,B 0,C 180,E1 -1080.677,E2 -1080.677} C_VEL
LIN {X 0,Y 594.247,Z 429.096,A -85,B 0,C 180,E1 -1082.033,E2 -1082.033} C_VEL
LIN {X 0,Y 594.278,Z 425.913,A -85,B 0,C 180,E1 -1083.05,E2 -1083.05} C_VEL
LIN {X 0,Y 594.262,Z 421.675,A -85,B 0,C 180,E1 -1084.069,E2 -1084.069} C_VEL
LIN {X 0,Y 594.263,Z 416.256,A -85,B 0,C 180,E1 -1085.089,E2 -1085.089} C_VEL
LIN {X 0,Y 594.329,Z 409.475,A -85,B 0,C 180,E1 -1086.109,E2 -1086.109} C_VEL
LIN {X 0,Y 594.357,Z 401.087,A -85,B 0,C 180,E1 -1087.132,E2 -1087.132} C_VEL
LIN {X 0,Y 594.389,Z 392.427,A -85,B 0,C 180,E1 -1087.986,E2 -1087.986} C_VEL
LIN {X 0,Y 594.44,Z 381.765,A -85,B 0,C 180,E1 -1088.841,E2 -1088.841} C_VEL
LIN {X 0,Y 594.498,Z 371.125,A -85,B 0,C 180,E1 -1089.526,E2 -1089.526} C_VEL
LIN {X 0,Y 594.572,Z 359.326,A -85,B 0,C 180,E1 -1090.127,E2 -1090.127} C_VEL
LIN {X 0,Y 594.598,Z 346.993,A -85,B 0,C 180,E1 -1090.6,E2 -1090.6} C_VEL
LIN {X 0,Y 594.602,Z 334.235,A -85,B 0,C 180,E1 -1090.945,E2 -1090.945} C_VEL
LIN {X 0,Y 594.648,Z 319.627,A -85,B 0,C 180,E1 -1091.175,E2 -1091.175} C_VEL
LIN {X 0,Y 594.643,Z 224.715,A -85,B 0,C 180,E1 -1092.326,E2 -1092.326} C_VEL
LIN {X 0,Y 594.309,Z 222.561,A -85,B 0,C 180,E1 -1092.377,E2 -1092.377} C_VEL
LIN {X 0,Y 594.423,Z 207.461,A -85,B 0,C 180,E1 -1095.077,E2 -1095.077} C_VEL
LIN {X 0,Y 594.415,Z 195.439,A -85,B 0,C 180,E1 -1097.281,E2 -1097.281} C_VEL
LIN {X 0,Y 594.373,Z 195.446,A -85,B 0,C 180,E1 -1100.054,E2 -1100.054} C_VEL
LIN {X 0,Y 594.359,Z 195.446,A -85,B 0,C 180,E1 -1102.967,E2 -1102.967} C_VEL
LIN {X 0,Y 594.364,Z 195.443,A -85,B 0,C 180,E1 -1105.194,E2 -1105.194} C_VEL
LIN {X 0,Y 594.373,Z 195.442,A -85,B 0,C 180,E1 -1107.523,E2 -1107.523} C_VEL
LIN {X 0,Y 594.376,Z 195.452,A -85,B 0,C 180,E1 -1110.325,E2 -1110.325} C_VEL
LIN {X 0,Y 594.381,Z 195.442,A -85,B 0,C 180,E1 -1112.95,E2 -1112.95} C_VEL
LIN {X 0,Y 594.352,Z 195.445,A -85,B 0,C 180,E1 -1115.409,E2 -1115.409} C_VEL
LIN {X 0,Y 594.389,Z 195.446,A -85,B 0,C 180,E1 -1117.941,E2 -1117.941} C_VEL
LIN {X 0,Y 594.375,Z 195.443,A -85,B 0,C 180,E1 -1120.821,E2 -1120.821} C_VEL
LIN {X 0,Y 594.356,Z 195.444,A -85,B 0,C 180,E1 -1123.301,E2 -1123.301} C_VEL
LIN {X 0,Y 594.366,Z 195.452,A -85,B 0,C 180,E1 -1126.161,E2 -1126.161} C_VEL
LIN {X 0,Y 594.374,Z 195.442,A -85,B 0,C 180,E1 -1129.179,E2 -1129.179} C_VEL
LIN {X 0,Y 594.383,Z 195.45,A -85,B 0,C 180,E1 -1132.058,E2 -1132.058} C_VEL
LIN {X 0,Y 594.351,Z 195.445,A -85,B 0,C 180,E1 -1134.677,E2 -1134.677} C_VEL
LIN {X 0,Y 594.38,Z 195.442,A -85,B 0,C 180,E1 -1137.089,E2 -1137.089} C_VEL
LIN {X 0,Y 594.39,Z 195.447,A -85,B 0,C 180,E1 -1139.672,E2 -1139.672} C_VEL
LIN {X 0,Y 594.38,Z 195.442,A -85,B 0,C 180,E1 -1142.539,E2 -1142.539} C_VEL
LIN {X 0,Y 594.404,Z 195.445,A -85,B 0,C 180,E1 -1145.564,E2 -1145.564} C_VEL
LIN {X 0,Y 594.381,Z 195.477,A -85,B 0,C 180,E1 -1146.572,E2 -1146.572} C_VEL
LIN {X 0,Y 594.792,Z 199.654,A -85,B 0,C 180,E1 -1147.167,E2 -1147.167} C_VEL
LIN {X 0,Y 594.679,Z 218.745,A -85,B 0,C 180,E1 -1149.776,E2 -1149.776} C_VEL
LIN {X 0,Y 594.57,Z 240.018,A -85,B 0,C 180,E1 -1152.634,E2 -1152.634} C_VEL
LIN {X 0,Y 594.451,Z 259.963,A -85,B 0,C 180,E1 -1155.274,E2 -1155.274} C_VEL
LIN {X 0,Y 594.434,Z 270.433,A -85,B 0,C 180,E1 -1156.648,E2 -1156.648} C_VEL
LIN {X 0,Y 594.729,Z 276.45,A -85,B 0,C 180,E1 -1156.742,E2 -1156.742} C_VEL
LIN {X 0,Y 594.665,Z 378.908,A -85,B 0,C 180,E1 -1157.998,E2 -1157.998} C_VEL
LIN {X 0,Y 594.634,Z 392.189,A -85,B 0,C 180,E1 -1158.3,E2 -1158.3} C_VEL
LIN {X 0,Y 594.599,Z 404.416,A -85,B 0,C 180,E1 -1158.713,E2 -1158.713} C_VEL
LIN {X 0,Y 594.528,Z 416.619,A -85,B 0,C 180,E1 -1159.269,E2 -1159.269} C_VEL
LIN {X 0,Y 594.48,Z 428.19,A -85,B 0,C 180,E1 -1159.957,E2 -1159.957} C_VEL
LIN {X 0,Y 594.414,Z 438.588,A -85,B 0,C 180,E1 -1160.729,E2 -1160.729} C_VEL
LIN {X 0,Y 594.383,Z 447.105,A -85,B 0,C 180,E1 -1161.5,E2 -1161.5} C_VEL
LIN {X 0,Y 594.347,Z 454.954,A -85,B 0,C 180,E1 -1162.355,E2 -1162.355} C_VEL
LIN {X 0,Y 594.283,Z 462.81,A -85,B 0,C 180,E1 -1163.408,E2 -1163.408} C_VEL
LIN {X 0,Y 594.289,Z 469.676,A -85,B 0,C 180,E1 -1164.571,E2 -1164.571} C_VEL
LIN {X 0,Y 594.27,Z 474.368,A -85,B 0,C 180,E1 -1165.591,E2 -1165.591} C_VEL
LIN {X 0,Y 594.267,Z 477.955,A -85,B 0,C 180,E1 -1166.609,E2 -1166.609} C_VEL
LIN {X 0,Y 594.226,Z 479.808,A -85,B 0,C 180,E1 -1167.288,E2 -1167.288} C_VEL
LIN {X 0,Y 594.242,Z 481.2,A -85,B 0,C 180,E1 -1167.966,E2 -1167.966} C_VEL
LIN {X 0,Y 594.239,Z 482.784,A -85,B 0,C 180,E1 -1169.322,E2 -1169.322} C_VEL
LIN {X 0,Y 594.236,Z 483,A -85,B 0,C 180,E1 -1169.999,E2 -1169.999} C_VEL
LIN {X 0,Y 594.247,Z 482.186,A -85,B 0,C 180,E1 -1171.355,E2 -1171.355} C_VEL
LIN {X 0,Y 594.242,Z 481.202,A -85,B 0,C 180,E1 -1172.033,E2 -1172.033} C_VEL
LIN {X 0,Y 594.226,Z 479.811,A -85,B 0,C 180,E1 -1172.711,E2 -1172.711} C_VEL
LIN {X 0,Y 594.289,Z 476.898,A -85,B 0,C 180,E1 -1173.729,E2 -1173.729} C_VEL
LIN {X 0,Y 594.241,Z 472.953,A -85,B 0,C 180,E1 -1174.748,E2 -1174.748} C_VEL
LIN {X 0,Y 594.305,Z 466.882,A -85,B 0,C 180,E1 -1175.938,E2 -1175.938} C_VEL
LIN {X 0,Y 594.311,Z 460.242,A -85,B 0,C 180,E1 -1176.961,E2 -1176.961} C_VEL
LIN {X 0,Y 594.359,Z 451.997,A -85,B 0,C 180,E1 -1177.986,E2 -1177.986} C_VEL
LIN {X 0,Y 594.382,Z 443.546,A -85,B 0,C 180,E1 -1178.841,E2 -1178.841} C_VEL
LIN {X 0,Y 594.434,Z 433.106,A -85,B 0,C 180,E1 -1179.699,E2 -1179.699} C_VEL
LIN {X 0,Y 594.483,Z 422.771,A -85,B 0,C 180,E1 -1180.386,E2 -1180.386} C_VEL
LIN {X 0,Y 594.557,Z 411.725,A -85,B 0,C 180,E1 -1180.973,E2 -1180.973} C_VEL
LIN {X 0,Y 594.577,Z 399.734,A -85,B 0,C 180,E1 -1181.464,E2 -1181.464} C_VEL
LIN {X 0,Y 594.625,Z 386.388,A -85,B 0,C 180,E1 -1181.85,E2 -1181.85} C_VEL
LIN {X 0,Y 594.693,Z 373.145,A -85,B 0,C 180,E1 -1182.086,E2 -1182.086} C_VEL
LIN {X 0,Y 594.624,Z 271.992,A -85,B 0,C 180,E1 -1183.315,E2 -1183.315} C_VEL
LIN {X 0,Y 594.433,Z 270.445,A -85,B 0,C 180,E1 -1183.35,E2 -1183.35} C_VEL
LIN {X 0,Y 594.536,Z 248.008,A -85,B 0,C 180,E1 -1186.304,E2 -1186.304} C_VEL
LIN {X 0,Y 594.623,Z 227.098,A -85,B 0,C 180,E1 -1189.097,E2 -1189.097} C_VEL
LIN {X 0,Y 594.773,Z 206.79,A -85,B 0,C 180,E1 -1191.851,E2 -1191.851} C_VEL
LIN {X 0,Y 594.748,Z 197.483,A -85,B 0,C 180,E1 -1193.135,E2 -1193.135} C_VEL
LIN {X 0,Y 594.351,Z 195.45,A -85,B 0,C 180,E1 -1193.451,E2 -1193.451} C_VEL
LIN {X 0,Y 594.365,Z 195.452,A -85,B 0,C 180,E1 -1196.018,E2 -1196.018} C_VEL
LIN {X 0,Y 594.373,Z 195.442,A -85,B 0,C 180,E1 -1198.956,E2 -1198.956} C_VEL
LIN {X 0,Y 594.372,Z 195.447,A -85,B 0,C 180,E1 -1201.641,E2 -1201.641} C_VEL
LIN {X 0,Y 594.364,Z 195.443,A -85,B 0,C 180,E1 -1204.58,E2 -1204.58} C_VEL
LIN {X 0,Y 594.381,Z 195.448,A -85,B 0,C 180,E1 -1207.607,E2 -1207.607} C_VEL
LIN {X 0,Y 594.353,Z 195.444,A -85,B 0,C 180,E1 -1210.567,E2 -1210.567} C_VEL
LIN {X 0,Y 594.353,Z 195.449,A -85,B 0,C 180,E1 -1213.299,E2 -1213.299} C_VEL
LIN {X 0,Y 594.335,Z 195.448,A -85,B 0,C 180,E1 -1216.162,E2 -1216.162} C_VEL
LIN {X 0,Y 594.358,Z 195.443,A -85,B 0,C 180,E1 -1218.534,E2 -1218.534} C_VEL
LIN {X 0,Y 594.36,Z 195.452,A -85,B 0,C 180,E1 -1221.297,E2 -1221.297} C_VEL
LIN {X 0,Y 594.336,Z 195.448,A -85,B 0,C 180,E1 -1223.754,E2 -1223.754} C_VEL
LIN {X 0,Y 594.34,Z 195.445,A -85,B 0,C 180,E1 -1226.236,E2 -1226.236} C_VEL
LIN {X 0,Y 594.352,Z 195.446,A -85,B 0,C 180,E1 -1228.649,E2 -1228.649} C_VEL
LIN {X 0,Y 594.365,Z 195.451,A -85,B 0,C 180,E1 -1231.043,E2 -1231.043} C_VEL
LIN {X 0,Y 594.36,Z 195.449,A -85,B 0,C 180,E1 -1233.299,E2 -1233.299} C_VEL
LIN {X 0,Y 594.327,Z 195.448,A -85,B 0,C 180,E1 -1236.293,E2 -1236.293} C_VEL
LIN {X 0,Y 594.368,Z 195.446,A -85,B 0,C 180,E1 -1239.223,E2 -1239.223} C_VEL
LIN {X 0,Y 594.311,Z 195.45,A -85,B 0,C 180,E1 -1242.094,E2 -1242.094} C_VEL
LIN {X 0,Y 594.327,Z 195.449,A -85,B 0,C 180,E1 -1244.218,E2 -1244.218} C_VEL
LIN {X 0,Y 594.317,Z 195.452,A -85,B 0,C 180,E1 -1247.016,E2 -1247.016} C_VEL
LIN {X 0,Y 594.339,Z 195.448,A -85,B 0,C 180,E1 -1249.094,E2 -1249.094} C_VEL
LIN {X 0,Y 594.338,Z 195.447,A -85,B 0,C 180,E1 -1251.842,E2 -1251.842} C_VEL
LIN {X 0,Y 594.376,Z 195.448,A -85,B 0,C 180,E1 -1254.572,E2 -1254.572} C_VEL
LIN {X 0,Y 594.365,Z 195.442,A -85,B 0,C 180,E1 -1257.289,E2 -1257.289} C_VEL
LIN {X 0,Y 594.394,Z 195.444,A -85,B 0,C 180,E1 -1260,E2 -1260} C_VEL
LIN {X 0,Y 594.392,Z 195.44,A -85,B 0,C 180,E1 -1262.711,E2 -1262.711} C_VEL
LIN {X 0,Y 594.357,Z 195.444,A -85,B 0,C 180,E1 -1265.428,E2 -1265.428} C_VEL
LIN {X 0,Y 594.403,Z 195.445,A -85,B 0,C 180,E1 -1268.157,E2 -1268.157} C_VEL
LIN {X 0,Y 594.362,Z 195.442,A -85,B 0,C 180,E1 -1271.065,E2 -1271.065} C_VEL
LIN {X 0,Y 594.366,Z 195.449,A -85,B 0,C 180,E1 -1273.68,E2 -1273.68} C_VEL
LIN {X 0,Y 594.344,Z 195.448,A -85,B 0,C 180,E1 -1275.325,E2 -1275.325} C_VEL
LIN {X 0,Y 593.674,Z 195.537,A -85,B 0,C 180,E1 -1275.891,E2 -1275.891} C_VEL
LIN {X 0,Y 590.811,Z 195.896,A -85,B 0,C 180,E1 -1276.809,E2 -1276.809} C_VEL
LIN {X 0,Y 588.4,Z 196.193,A -85,B 0,C 180,E1 -1277.547,E2 -1277.547} C_VEL
LIN {X 0,Y 587.375,Z 196.317,A -85,B 0,C 180,E1 -1278.118,E2 -1278.118} C_VEL
LIN {X 0,Y 587.297,Z 196.324,A -85,B 0,C 180,E1 -1278.311,E2 -1278.311} C_VEL
LIN {X 0,Y 587.323,Z 196.321,A -85,B 0,C 180,E1 -1281.038,E2 -1281.038} C_VEL
LIN {X 0,Y 587.316,Z 196.325,A -85,B 0,C 180,E1 -1283.259,E2 -1283.259} C_VEL
LIN {X 0,Y 587.33,Z 196.328,A -85,B 0,C 180,E1 -1285.517,E2 -1285.517} C_VEL
LIN {X 0,Y 587.338,Z 196.322,A -85,B 0,C 180,E1 -1287.819,E2 -1287.819} C_VEL
LIN {X 0,Y 587.335,Z 196.318,A -85,B 0,C 180,E1 -1290.511,E2 -1290.511} C_VEL
LIN {X 0,Y 587.331,Z 196.327,A -85,B 0,C 180,E1 -1293.397,E2 -1293.397} C_VEL
LIN {X 0,Y 587.314,Z 196.323,A -85,B 0,C 180,E1 -1295.899,E2 -1295.899} C_VEL
LIN {X 0,Y 587.328,Z 196.32,A -85,B 0,C 180,E1 -1298.48,E2 -1298.48} C_VEL
LIN {X 0,Y 587.333,Z 196.327,A -85,B 0,C 180,E1 -1301.158,E2 -1301.158} C_VEL
LIN {X 0,Y 587.332,Z 196.319,A -85,B 0,C 180,E1 -1304.115,E2 -1304.115} C_VEL
LIN {X 0,Y 587.316,Z 196.33,A -85,B 0,C 180,E1 -1306.995,E2 -1306.995} C_VEL
LIN {X 0,Y 587.312,Z 196.321,A -85,B 0,C 180,E1 -1309.747,E2 -1309.747} C_VEL
LIN {X 0,Y 587.344,Z 196.322,A -85,B 0,C 180,E1 -1312.393,E2 -1312.393} C_VEL
LIN {X 0,Y 587.36,Z 196.316,A -85,B 0,C 180,E1 -1315.781,E2 -1315.781} C_VEL
LIN {X 0,Y 587.393,Z 196.451,A -85,B 0,C 180,E1 -1317.796,E2 -1317.796} C_VEL
LIN {X 0,Y 587.383,Z 210.813,A -85,B 0,C 180,E1 -1320.427,E2 -1320.427} C_VEL
LIN {X 0,Y 587.292,Z 222.553,A -85,B 0,C 180,E1 -1322.55,E2 -1322.55} C_VEL
LIN {X 0,Y 587.855,Z 226.911,A -85,B 0,C 180,E1 -1322.635,E2 -1322.635} C_VEL
LIN {X 0,Y 587.681,Z 329.291,A -85,B 0,C 180,E1 -1323.906,E2 -1323.906} C_VEL
LIN {X 0,Y 587.602,Z 342.525,A -85,B 0,C 180,E1 -1324.212,E2 -1324.212} C_VEL
LIN {X 0,Y 587.585,Z 354.865,A -85,B 0,C 180,E1 -1324.638,E2 -1324.638} C_VEL
LIN {X 0,Y 587.546,Z 366.064,A -85,B 0,C 180,E1 -1325.157,E2 -1325.157} C_VEL
LIN {X 0,Y 587.403,Z 377.443,A -85,B 0,C 180,E1 -1325.828,E2 -1325.828} C_VEL
LIN {X 0,Y 587.378,Z 388.467,A -85,B 0,C 180,E1 -1326.651,E2 -1326.651} C_VEL
LIN {X 0,Y 587.327,Z 397.546,A -85,B 0,C 180,E1 -1327.487,E2 -1327.487} C_VEL
LIN {X 0,Y 587.273,Z 405.778,A -85,B 0,C 180,E1 -1328.409,E2 -1328.409} C_VEL
LIN {X 0,Y 587.218,Z 413.698,A -85,B 0,C 180,E1 -1329.509,E2 -1329.509} C_VEL
LIN {X 0,Y 587.19,Z 419.003,A -85,B 0,C 180,E1 -1330.421,E2 -1330.421} C_VEL
LIN {X 0,Y 587.174,Z 424.068,A -85,B 0,C 180,E1 -1331.508,E2 -1331.508} C_VEL
LIN {X 0,Y 587.162,Z 427.882,A -85,B 0,C 180,E1 -1332.589,E2 -1332.589} C_VEL
LIN {X 0,Y 587.168,Z 429.821,A -85,B 0,C 180,E1 -1333.307,E2 -1333.307} C_VEL
LIN {X 0,Y 587.139,Z 431.253,A -85,B 0,C 180,E1 -1334.021,E2 -1334.021} C_VEL
LIN {X 0,Y 587.125,Z 432.251,A -85,B 0,C 180,E1 -1334.732,E2 -1334.732} C_VEL
LIN {X 0,Y 587.161,Z 432.955,A -85,B 0,C 180,E1 -1335.821,E2 -1335.821} C_VEL
LIN {X 0,Y 587.146,Z 432.699,A -85,B 0,C 180,E1 -1336.855,E2 -1336.855} C_VEL
LIN {X 0,Y 587.16,Z 432.022,A -85,B 0,C 180,E1 -1337.559,E2 -1337.559} C_VEL
LIN {X 0,Y 587.155,Z 430.925,A -85,B 0,C 180,E1 -1338.26,E2 -1338.26} C_VEL
LIN {X 0,Y 587.168,Z 429.373,A -85,B 0,C 180,E1 -1338.96,E2 -1338.96} C_VEL
LIN {X 0,Y 587.179,Z 426.243,A -85,B 0,C 180,E1 -1340.006,E2 -1340.006} C_VEL
LIN {X 0,Y 587.187,Z 422.054,A -85,B 0,C 180,E1 -1341.049,E2 -1341.049} C_VEL
LIN {X 0,Y 587.232,Z 415.673,A -85,B 0,C 180,E1 -1342.263,E2 -1342.263} C_VEL
LIN {X 0,Y 587.239,Z 408.093,A -85,B 0,C 180,E1 -1343.385,E2 -1343.385} C_VEL
LIN {X 0,Y 587.29,Z 400.107,A -85,B 0,C 180,E1 -1344.335,E2 -1344.335} C_VEL
LIN {X 0,Y 587.388,Z 391.277,A -85,B 0,C 180,E1 -1345.196,E2 -1345.196} C_VEL
LIN {X 0,Y 587.406,Z 381.652,A -85,B 0,C 180,E1 -1345.97,E2 -1345.97} C_VEL
LIN {X 0,Y 587.491,Z 371.068,A -85,B 0,C 180,E1 -1346.657,E2 -1346.657} C_VEL
LIN {X 0,Y 587.591,Z 359.364,A -85,B 0,C 180,E1 -1347.259,E2 -1347.259} C_VEL
LIN {X 0,Y 587.613,Z 347.279,A -85,B 0,C 180,E1 -1347.73,E2 -1347.73} C_VEL
LIN {X 0,Y 587.688,Z 334.845,A -85,B 0,C 180,E1 -1348.073,E2 -1348.073} C_VEL
LIN {X 0,Y 587.738,Z 322.248,A -85,B 0,C 180,E1 -1348.288,E2 -1348.288} C_VEL
LIN {X 0,Y 587.751,Z 225.305,A -85,B 0,C 180,E1 -1349.478,E2 -1349.478} C_VEL
LIN {X 0,Y 587.308,Z 222.611,A -85,B 0,C 180,E1 -1349.529,E2 -1349.529} C_VEL
LIN {X 0,Y 587.379,Z 208.647,A -85,B 0,C 180,E1 -1352.058,E2 -1352.058} C_VEL
LIN {X 0,Y 587.396,Z 197.405,A -85,B 0,C 180,E1 -1354.117,E2 -1354.117} C_VEL
LIN {X 0,Y 587.334,Z 196.322,A -85,B 0,C 180,E1 -1354.333,E2 -1354.333} C_VEL
LIN {X 0,Y 587.364,Z 196.317,A -85,B 0,C 180,E1 -1356.873,E2 -1356.873} C_VEL
LIN {X 0,Y 587.307,Z 196.327,A -85,B 0,C 180,E1 -1359.645,E2 -1359.645} C_VEL
LIN {X 0,Y 587.338,Z 196.322,A -85,B 0,C 180,E1 -1361.738,E2 -1361.738} C_VEL
LIN {X 0,Y 587.322,Z 196.322,A -85,B 0,C 180,E1 -1364.555,E2 -1364.555} C_VEL
LIN {X 0,Y 587.31,Z 196.327,A -85,B 0,C 180,E1 -1367.408,E2 -1367.408} C_VEL
LIN {X 0,Y 587.307,Z 196.325,A -85,B 0,C 180,E1 -1369.577,E2 -1369.577} C_VEL
LIN {X 0,Y 587.309,Z 196.323,A -85,B 0,C 180,E1 -1371.776,E2 -1371.776} C_VEL
LIN {X 0,Y 587.314,Z 196.326,A -85,B 0,C 180,E1 -1374.571,E2 -1374.571} C_VEL
LIN {X 0,Y 587.303,Z 196.33,A -85,B 0,C 180,E1 -1377.048,E2 -1377.048} C_VEL
LIN {X 0,Y 587.314,Z 196.323,A -85,B 0,C 180,E1 -1379.382,E2 -1379.382} C_VEL
LIN {X 0,Y 587.321,Z 196.321,A -85,B 0,C 180,E1 -1381.831,E2 -1381.831} C_VEL
LIN {X 0,Y 587.319,Z 196.326,A -85,B 0,C 180,E1 -1384.343,E2 -1384.343} C_VEL
LIN {X 0,Y 587.311,Z 196.329,A -85,B 0,C 180,E1 -1386.75,E2 -1386.75} C_VEL
LIN {X 0,Y 587.317,Z 196.321,A -85,B 0,C 180,E1 -1389.362,E2 -1389.362} C_VEL
LIN {X 0,Y 587.298,Z 196.328,A -85,B 0,C 180,E1 -1392.103,E2 -1392.103} C_VEL
LIN {X 0,Y 587.282,Z 196.327,A -85,B 0,C 180,E1 -1394.915,E2 -1394.915} C_VEL
LIN {X 0,Y 587.303,Z 196.328,A -85,B 0,C 180,E1 -1397.923,E2 -1397.923} C_VEL
LIN {X 0,Y 587.306,Z 196.326,A -85,B 0,C 180,E1 -1400.637,E2 -1400.637} C_VEL
LIN {X 0,Y 587.267,Z 196.328,A -85,B 0,C 180,E1 -1403.304,E2 -1403.304} C_VEL
LIN {X 0,Y 587.309,Z 196.328,A -85,B 0,C 180,E1 -1405.776,E2 -1405.776} C_VEL
LIN {X 0,Y 587.304,Z 196.328,A -85,B 0,C 180,E1 -1408.228,E2 -1408.228} C_VEL
LIN {X 0,Y 587.301,Z 196.323,A -85,B 0,C 180,E1 -1410.876,E2 -1410.876} C_VEL
LIN {X 0,Y 587.297,Z 196.333,A -85,B 0,C 180,E1 -1413.833,E2 -1413.833} C_VEL
LIN {X 0,Y 587.316,Z 196.327,A -85,B 0,C 180,E1 -1415.992,E2 -1415.992} C_VEL
LIN {X 0,Y 587.338,Z 196.32,A -85,B 0,C 180,E1 -1418.962,E2 -1418.962} C_VEL
LIN {X 0,Y 587.303,Z 196.343,A -85,B 0,C 180,E1 -1420.774,E2 -1420.774} C_VEL
LIN {X 0,Y 587.38,Z 206.249,A -85,B 0,C 180,E1 -1422.595,E2 -1422.595} C_VEL
LIN {X 0,Y 587.343,Z 221.973,A -85,B 0,C 180,E1 -1425.446,E2 -1425.446} C_VEL
LIN {X 0,Y 587.326,Z 222.67,A -85,B 0,C 180,E1 -1425.57,E2 -1425.57} C_VEL
LIN {X 0,Y 587.862,Z 228.018,A -85,B 0,C 180,E1 -1425.648,E2 -1425.648} C_VEL
LIN {X 0,Y 587.709,Z 329.508,A -85,B 0,C 180,E1 -1426.911,E2 -1426.911} C_VEL
LIN {X 0,Y 587.698,Z 342.687,A -85,B 0,C 180,E1 -1427.218,E2 -1427.218} C_VEL
LIN {X 0,Y 587.625,Z 355.203,A -85,B 0,C 180,E1 -1427.655,E2 -1427.655} C_VEL
LIN {X 0,Y 587.522,Z 366.503,A -85,B 0,C 180,E1 -1428.179,E2 -1428.179} C_VEL
LIN {X 0,Y 587.424,Z 378.382,A -85,B 0,C 180,E1 -1428.893,E2 -1428.893} C_VEL
LIN {X 0,Y 587.365,Z 388.541,A -85,B 0,C 180,E1 -1429.66,E2 -1429.66} C_VEL
LIN {X 0,Y 587.324,Z 397.948,A -85,B 0,C 180,E1 -1430.53,E2 -1430.53} C_VEL
LIN {X 0,Y 587.249,Z 407.045,A -85,B 0,C 180,E1 -1431.57,E2 -1431.57} C_VEL
LIN {X 0,Y 587.238,Z 414.324,A -85,B 0,C 180,E1 -1432.608,E2 -1432.608} C_VEL
LIN {X 0,Y 587.175,Z 420.125,A -85,B 0,C 180,E1 -1433.641,E2 -1433.641} C_VEL
LIN {X 0,Y 587.201,Z 424.045,A -85,B 0,C 180,E1 -1434.505,E2 -1434.505} C_VEL
LIN {X 0,Y 587.189,Z 427.705,A -85,B 0,C 180,E1 -1435.538,E2 -1435.538} C_VEL
LIN {X 0,Y 587.183,Z 430.369,A -85,B 0,C 180,E1 -1436.569,E2 -1436.569} C_VEL
LIN {X 0,Y 587.131,Z 431.639,A -85,B 0,C 180,E1 -1437.255,E2 -1437.255} C_VEL
LIN {X 0,Y 587.137,Z 432.484,A -85,B 0,C 180,E1 -1437.942,E2 -1437.942} C_VEL
LIN {X 0,Y 587.139,Z 432.945,A -85,B 0,C 180,E1 -1439.314,E2 -1439.314} C_VEL
LIN {X 0,Y 587.138,Z 432.606,A -85,B 0,C 180,E1 -1440,E2 -1440} C_VEL
LIN {X 0,Y 587.14,Z 431.843,A -85,B 0,C 180,E1 -1440.686,E2 -1440.686} C_VEL
LIN {X 0,Y 587.149,Z 429.129,A -85,B 0,C 180,E1 -1442.058,E2 -1442.058} C_VEL
LIN {X 0,Y 587.183,Z 425.957,A -85,B 0,C 180,E1 -1443.087,E2 -1443.087} C_VEL
LIN {X 0,Y 587.183,Z 421.73,A -85,B 0,C 180,E1 -1444.118,E2 -1444.118} C_VEL
LIN {X 0,Y 587.177,Z 416.322,A -85,B 0,C 180,E1 -1445.15,E2 -1445.15} C_VEL
LIN {X 0,Y 587.268,Z 409.55,A -85,B 0,C 180,E1 -1446.183,E2 -1446.183} C_VEL
LIN {X 0,Y 587.295,Z 401.189,A -85,B 0,C 180,E1 -1447.218,E2 -1447.218} C_VEL
LIN {X 0,Y 587.384,Z 390.607,A -85,B 0,C 180,E1 -1448.255,E2 -1448.255} C_VEL
LIN {X 0,Y 587.442,Z 380.697,A -85,B 0,C 180,E1 -1449.034,E2 -1449.034} C_VEL
LIN {X 0,Y 587.529,Z 369.838,A -85,B 0,C 180,E1 -1449.727,E2 -1449.727} C_VEL
LIN {X 0,Y 587.61,Z 356.588,A -85,B 0,C 180,E1 -1450.379,E2 -1450.379} C_VEL
LIN {X 0,Y 587.666,Z 344.618,A -85,B 0,C 180,E1 -1450.813,E2 -1450.813} C_VEL
LIN {X 0,Y 587.692,Z 331.927,A -85,B 0,C 180,E1 -1451.135,E2 -1451.135} C_VEL
LIN {X 0,Y 587.726,Z 312.798,A -85,B 0,C 180,E1 -1451.404,E2 -1451.404} C_VEL
LIN {X 0,Y 587.715,Z 225.355,A -85,B 0,C 180,E1 -1452.478,E2 -1452.478} C_VEL
LIN {X 0,Y 587.29,Z 222.627,A -85,B 0,C 180,E1 -1452.527,E2 -1452.527} C_VEL
LIN {X 0,Y 587.409,Z 207.529,A -85,B 0,C 180,E1 -1455.261,E2 -1455.261} C_VEL
LIN {X 0,Y 587.382,Z 196.316,A -85,B 0,C 180,E1 -1457.321,E2 -1457.321} C_VEL
LIN {X 0,Y 587.331,Z 196.328,A -85,B 0,C 180,E1 -1460.305,E2 -1460.305} C_VEL
LIN {X 0,Y 587.315,Z 196.322,A -85,B 0,C 180,E1 -1463.259,E2 -1463.259} C_VEL
LIN {X 0,Y 587.325,Z 196.32,A -85,B 0,C 180,E1 -1465.517,E2 -1465.517} C_VEL
LIN {X 0,Y 587.345,Z 196.32,A -85,B 0,C 180,E1 -1467.818,E2 -1467.818} C_VEL
LIN {X 0,Y 587.331,Z 196.326,A -85,B 0,C 180,E1 -1470.508,E2 -1470.508} C_VEL
LIN {X 0,Y 587.341,Z 196.318,A -85,B 0,C 180,E1 -1473.111,E2 -1473.111} C_VEL
LIN {X 0,Y 587.299,Z 196.324,A -85,B 0,C 180,E1 -1475.537,E2 -1475.537} C_VEL
LIN {X 0,Y 587.343,Z 196.322,A -85,B 0,C 180,E1 -1477.838,E2 -1477.838} C_VEL
LIN {X 0,Y 587.314,Z 196.33,A -85,B 0,C 180,E1 -1480.254,E2 -1480.254} C_VEL
LIN {X 0,Y 587.308,Z 196.322,A -85,B 0,C 180,E1 -1483.117,E2 -1483.117} C_VEL
LIN {X 0,Y 587.319,Z 196.33,A -85,B 0,C 180,E1 -1486.048,E2 -1486.048} C_VEL
LIN {X 0,Y 587.337,Z 196.318,A -85,B 0,C 180,E1 -1488.925,E2 -1488.925} C_VEL
LIN {X 0,Y 587.323,Z 196.323,A -85,B 0,C 180,E1 -1491.519,E2 -1491.519} C_VEL
LIN {X 0,Y 587.292,Z 196.332,A -85,B 0,C 180,E1 -1494.099,E2 -1494.099} C_VEL
LIN {X 0,Y 587.338,Z 196.32,A -85,B 0,C 180,E1 -1496.603,E2 -1496.603} C_VEL
LIN {X 0,Y 587.339,Z 196.323,A -85,B 0,C 180,E1 -1499.49,E2 -1499.49} C_VEL
LIN {X 0,Y 587.309,Z 196.328,A -85,B 0,C 180,E1 -1502.18,E2 -1502.18} C_VEL
LIN {X 0,Y 587.355,Z 196.32,A -85,B 0,C 180,E1 -1505.241,E2 -1505.241} C_VEL
LIN {X 0,Y 587.341,Z 196.369,A -85,B 0,C 180,E1 -1506.414,E2 -1506.414} C_VEL
LIN {X 0,Y 587.889,Z 200.49,A -85,B 0,C 180,E1 -1507.001,E2 -1507.001} C_VEL
LIN {X 0,Y 587.754,Z 218.745,A -85,B 0,C 180,E1 -1509.527,E2 -1509.527} C_VEL
LIN {X 0,Y 587.581,Z 241.348,A -85,B 0,C 180,E1 -1512.6,E2 -1512.6} C_VEL
LIN {X 0,Y 587.459,Z 259.963,A -85,B 0,C 180,E1 -1515.095,E2 -1515.095} C_VEL
LIN {X 0,Y 587.402,Z 270.433,A -85,B 0,C 180,E1 -1516.485,E2 -1516.485} C_VEL
LIN {X 0,Y 587.841,Z 274.661,A -85,B 0,C 180,E1 -1516.562,E2 -1516.562} C_VEL
LIN {X 0,Y 587.726,Z 378.908,A -85,B 0,C 180,E1 -1517.854,E2 -1517.854} C_VEL
LIN {X 0,Y 587.686,Z 392.189,A -85,B 0,C 180,E1 -1518.16,E2 -1518.16} C_VEL
LIN {X 0,Y 587.63,Z 404.585,A -85,B 0,C 180,E1 -1518.584,E2 -1518.584} C_VEL
LIN {X 0,Y 587.53,Z 416.618,A -85,B 0,C 180,E1 -1519.14,E2 -1519.14} C_VEL
LIN {X 0,Y 587.467,Z 428.192,A -85,B 0,C 180,E1 -1519.836,E2 -1519.836} C_VEL
LIN {X 0,Y 587.366,Z 438.589,A -85,B 0,C 180,E1 -1520.617,E2 -1520.617} C_VEL
LIN {X 0,Y 587.322,Z 447.105,A -85,B 0,C 180,E1 -1521.397,E2 -1521.397} C_VEL
LIN {X 0,Y 587.274,Z 454.954,A -85,B 0,C 180,E1 -1522.262,E2 -1522.262} C_VEL
LIN {X 0,Y 587.231,Z 461.464,A -85,B 0,C 180,E1 -1523.126,E2 -1523.126} C_VEL
LIN {X 0,Y 587.237,Z 467.863,A -85,B 0,C 180,E1 -1524.161,E2 -1524.161} C_VEL
LIN {X 0,Y 587.147,Z 472.946,A -85,B 0,C 180,E1 -1525.193,E2 -1525.193} C_VEL
LIN {X 0,Y 587.213,Z 476.894,A -85,B 0,C 180,E1 -1526.225,E2 -1526.225} C_VEL
LIN {X 0,Y 587.132,Z 479.808,A -85,B 0,C 180,E1 -1527.255,E2 -1527.255} C_VEL
LIN {X 0,Y 587.141,Z 481.199,A -85,B 0,C 180,E1 -1527.941,E2 -1527.941} C_VEL
LIN {X 0,Y 587.14,Z 482.784,A -85,B 0,C 180,E1 -1529.313,E2 -1529.313} C_VEL
LIN {X 0,Y 587.137,Z 483,A -85,B 0,C 180,E1 -1529.999,E2 -1529.999} C_VEL
LIN {X 0,Y 587.147,Z 482.186,A -85,B 0,C 180,E1 -1531.371,E2 -1531.371} C_VEL
LIN {X 0,Y 587.141,Z 481.201,A -85,B 0,C 180,E1 -1532.057,E2 -1532.057} C_VEL
LIN {X 0,Y 587.132,Z 479.81,A -85,B 0,C 180,E1 -1532.744,E2 -1532.744} C_VEL
LIN {X 0,Y 587.213,Z 476.898,A -85,B 0,C 180,E1 -1533.774,E2 -1533.774} C_VEL
LIN {X 0,Y 587.147,Z 472.953,A -85,B 0,C 180,E1 -1534.806,E2 -1534.806} C_VEL
LIN {X 0,Y 587.218,Z 466.882,A -85,B 0,C 180,E1 -1536.01,E2 -1536.01} C_VEL
LIN {X 0,Y 587.246,Z 460.243,A -85,B 0,C 180,E1 -1537.045,E2 -1537.045} C_VEL
LIN {X 0,Y 587.299,Z 451.997,A -85,B 0,C 180,E1 -1538.082,E2 -1538.082} C_VEL
LIN {X 0,Y 587.343,Z 443.547,A -85,B 0,C 180,E1 -1538.948,E2 -1538.948} C_VEL
LIN {X 0,Y 587.421,Z 433.107,A -85,B 0,C 180,E1 -1539.815,E2 -1539.815} C_VEL
LIN {X 0,Y 587.487,Z 422.769,A -85,B 0,C 180,E1 -1540.511,E2 -1540.511} C_VEL
LIN {X 0,Y 587.581,Z 410.832,A -85,B 0,C 180,E1 -1541.148,E2 -1541.148} C_VEL
LIN {X 0,Y 587.626,Z 398.626,A -85,B 0,C 180,E1 -1541.639,E2 -1541.639} C_VEL
LIN {X 0,Y 587.703,Z 385.473,A -85,B 0,C 180,E1 -1542.013,E2 -1542.013} C_VEL
LIN {X 0,Y 587.776,Z 373.145,A -85,B 0,C 180,E1 -1542.231,E2 -1542.231} C_VEL
LIN {X 0,Y 587.72,Z 272.551,A -85,B 0,C 180,E1 -1543.467,E2 -1543.467} C_VEL
LIN {X 0,Y 587.404,Z 270.279,A -85,B 0,C 180,E1 -1543.535,E2 -1543.535} C_VEL
LIN {X 0,Y 587.551,Z 248.008,A -85,B 0,C 180,E1 -1546.503,E2 -1546.503} C_VEL
LIN {X 0,Y 587.668,Z 227.451,A -85,B 0,C 180,E1 -1549.283,E2 -1549.283} C_VEL
LIN {X 0,Y 587.864,Z 206.79,A -85,B 0,C 180,E1 -1552.121,E2 -1552.121} C_VEL
LIN {X 0,Y 587.798,Z 198.797,A -85,B 0,C 180,E1 -1553.238,E2 -1553.238} C_VEL
LIN {X 0,Y 587.328,Z 196.326,A -85,B 0,C 180,E1 -1553.631,E2 -1553.631} C_VEL
LIN {X 0,Y 587.326,Z 196.328,A -85,B 0,C 180,E1 -1556.278,E2 -1556.278} C_VEL
LIN {X 0,Y 587.342,Z 196.318,A -85,B 0,C 180,E1 -1559.132,E2 -1559.132} C_VEL
LIN {X 0,Y 587.336,Z 196.327,A -85,B 0,C 180,E1 -1561.834,E2 -1561.834} C_VEL
LIN {X 0,Y 587.337,Z 196.32,A -85,B 0,C 180,E1 -1564.346,E2 -1564.346} C_VEL
LIN {X 0,Y 587.336,Z 196.325,A -85,B 0,C 180,E1 -1567.607,E2 -1567.607} C_VEL
LIN {X 0,Y 587.3,Z 196.325,A -85,B 0,C 180,E1 -1570.254,E2 -1570.254} C_VEL
LIN {X 0,Y 587.294,Z 196.325,A -85,B 0,C 180,E1 -1573.116,E2 -1573.116} C_VEL
LIN {X 0,Y 587.291,Z 196.326,A -85,B 0,C 180,E1 -1576.046,E2 -1576.046} C_VEL
LIN {X 0,Y 587.322,Z 196.321,A -85,B 0,C 180,E1 -1578.925,E2 -1578.925} C_VEL
LIN {X 0,Y 587.307,Z 196.329,A -85,B 0,C 180,E1 -1581.519,E2 -1581.519} C_VEL
LIN {X 0,Y 587.279,Z 196.324,A -85,B 0,C 180,E1 -1584.099,E2 -1584.099} C_VEL
LIN {X 0,Y 587.322,Z 196.324,A -85,B 0,C 180,E1 -1586.889,E2 -1586.889} C_VEL
LIN {X 0,Y 587.298,Z 196.326,A -85,B 0,C 180,E1 -1589.495,E2 -1589.495} C_VEL
LIN {X 0,Y 587.286,Z 196.328,A -85,B 0,C 180,E1 -1591.401,E2 -1591.401} C_VEL
LIN {X 0,Y 587.285,Z 196.325,A -85,B 0,C 180,E1 -1593.832,E2 -1593.832} C_VEL
LIN {X 0,Y 587.285,Z 196.33,A -85,B 0,C 180,E1 -1596.74,E2 -1596.74} C_VEL
LIN {X 0,Y 587.292,Z 196.323,A -85,B 0,C 180,E1 -1599.694,E2 -1599.694} C_VEL
LIN {X 0,Y 587.263,Z 196.327,A -85,B 0,C 180,E1 -1601.871,E2 -1601.871} C_VEL
LIN {X 0,Y 587.278,Z 196.326,A -85,B 0,C 180,E1 -1604.024,E2 -1604.024} C_VEL
LIN {X 0,Y 587.316,Z 196.321,A -85,B 0,C 180,E1 -1606.153,E2 -1606.153} C_VEL
LIN {X 0,Y 587.327,Z 196.323,A -85,B 0,C 180,E1 -1608.962,E2 -1608.962} C_VEL
LIN {X 0,Y 587.304,Z 196.323,A -85,B 0,C 180,E1 -1611.744,E2 -1611.744} C_VEL
LIN {X 0,Y 587.339,Z 196.325,A -85,B 0,C 180,E1 -1614.507,E2 -1614.507} C_VEL
LIN {X 0,Y 587.335,Z 196.318,A -85,B 0,C 180,E1 -1617.257,E2 -1617.257} C_VEL
LIN {X 0,Y 587.364,Z 196.32,A -85,B 0,C 180,E1 -1620,E2 -1620} C_VEL
LIN {X 0,Y 587.356,Z 196.315,A -85,B 0,C 180,E1 -1622.744,E2 -1622.744} C_VEL
LIN {X 0,Y 587.326,Z 196.32,A -85,B 0,C 180,E1 -1625.493,E2 -1625.493} C_VEL
LIN {X 0,Y 587.355,Z 196.321,A -85,B 0,C 180,E1 -1628.256,E2 -1628.256} C_VEL
LIN {X 0,Y 587.34,Z 196.316,A -85,B 0,C 180,E1 -1631.134,E2 -1631.134} C_VEL
LIN {X 0,Y 587.357,Z 196.319,A -85,B 0,C 180,E1 -1634.261,E2 -1634.261} C_VEL
LIN {X 0,Y 587.333,Z 196.321,A -85,B 0,C 180,E1 -1637.407,E2 -1637.407} C_VEL
LIN {X 0,Y 587.297,Z 196.324,A -85,B 0,C 180,E1 -1638.311,E2 -1638.311} C_VEL
LIN {X 0,Y 586.653,Z 196.404,A -85,B 0,C 180,E1 -1638.883,E2 -1638.883} C_VEL
LIN {X 0,Y 583.831,Z 196.763,A -85,B 0,C 180,E1 -1639.811,E2 -1639.811} C_VEL
LIN {X 0,Y 581.423,Z 197.064,A -85,B 0,C 180,E1 -1640.558,E2 -1640.558} C_VEL
LIN {X 0,Y 580.371,Z 197.192,A -85,B 0,C 180,E1 -1641.135,E2 -1641.135} C_VEL
LIN {X 0,Y 580.275,Z 197.202,A -85,B 0,C 180,E1 -1641.33,E2 -1641.33} C_VEL
LIN {X 0,Y 580.295,Z 197.195,A -85,B 0,C 180,E1 -1644.317,E2 -1644.317} C_VEL
LIN {X 0,Y 580.28,Z 197.206,A -85,B 0,C 180,E1 -1647.403,E2 -1647.403} C_VEL
LIN {X 0,Y 580.281,Z 197.201,A -85,B 0,C 180,E1 -1649.773,E2 -1649.773} C_VEL
LIN {X 0,Y 580.295,Z 197.196,A -85,B 0,C 180,E1 -1652.201,E2 -1652.201} C_VEL
LIN {X 0,Y 580.284,Z 197.198,A -85,B 0,C 180,E1 -1654.697,E2 -1654.697} C_VEL
LIN {X 0,Y 580.296,Z 197.204,A -85,B 0,C 180,E1 -1657.269,E2 -1657.269} C_VEL
LIN {X 0,Y 580.293,Z 197.197,A -85,B 0,C 180,E1 -1660.272,E2 -1660.272} C_VEL
LIN {X 0,Y 580.278,Z 197.202,A -85,B 0,C 180,E1 -1662.707,E2 -1662.707} C_VEL
LIN {X 0,Y 580.268,Z 197.2,A -85,B 0,C 180,E1 -1665.61,E2 -1665.61} C_VEL
LIN {X 0,Y 580.297,Z 197.197,A -85,B 0,C 180,E1 -1668.234,E2 -1668.234} C_VEL
LIN {X 0,Y 580.278,Z 197.205,A -85,B 0,C 180,E1 -1670.966,E2 -1670.966} C_VEL
LIN {X 0,Y 580.267,Z 197.2,A -85,B 0,C 180,E1 -1673.597,E2 -1673.597} C_VEL
LIN {X 0,Y 580.315,Z 197.196,A -85,B 0,C 180,E1 -1676.146,E2 -1676.146} C_VEL
LIN {X 0,Y 580.343,Z 197.305,A -85,B 0,C 180,E1 -1677.726,E2 -1677.726} C_VEL
LIN {X 0,Y 580.366,Z 209.727,A -85,B 0,C 180,E1 -1680.033,E2 -1680.033} C_VEL
LIN {X 0,Y 580.274,Z 222.621,A -85,B 0,C 180,E1 -1682.396,E2 -1682.396} C_VEL
LIN {X 0,Y 580.941,Z 228.25,A -85,B 0,C 180,E1 -1682.489,E2 -1682.489} C_VEL
LIN {X 0,Y 580.742,Z 329.45,A -85,B 0,C 180,E1 -1683.762,E2 -1683.762} C_VEL
LIN {X 0,Y 580.669,Z 342.495,A -85,B 0,C 180,E1 -1684.067,E2 -1684.067} C_VEL
LIN {X 0,Y 580.606,Z 354.96,A -85,B 0,C 180,E1 -1684.504,E2 -1684.504} C_VEL
LIN {X 0,Y 580.562,Z 366.166,A -85,B 0,C 180,E1 -1685.03,E2 -1685.03} C_VEL
LIN {X 0,Y 580.404,Z 377.243,A -85,B 0,C 180,E1 -1685.689,E2 -1685.689} C_VEL
LIN {X 0,Y 580.379,Z 387.393,A -85,B 0,C 180,E1 -1686.447,E2 -1686.447} C_VEL
LIN {X 0,Y 580.294,Z 397.586,A -85,B 0,C 180,E1 -1687.387,E2 -1687.387} C_VEL
LIN {X 0,Y 580.22,Z 405.815,A -85,B 0,C 180,E1 -1688.32,E2 -1688.32} C_VEL
LIN {X 0,Y 580.137,Z 413.726,A -85,B 0,C 180,E1 -1689.433,E2 -1689.433} C_VEL
LIN {X 0,Y 580.1,Z 419.969,A -85,B 0,C 180,E1 -1690.54,E2 -1690.54} C_VEL
LIN {X 0,Y 580.074,Z 424.817,A -85,B 0,C 180,E1 -1691.64,E2 -1691.64} C_VEL
LIN {X 0,Y 580.055,Z 428.438,A -85,B 0,C 180,E1 -1692.733,E2 -1692.733} C_VEL
LIN {X 0,Y 580.039,Z 430.958,A -85,B 0,C 180,E1 -1693.82,E2 -1693.82} C_VEL
LIN {X 0,Y 580.021,Z 432.053,A -85,B 0,C 180,E1 -1694.541,E2 -1694.541} C_VEL
LIN {X 0,Y 580.052,Z 432.944,A -85,B 0,C 180,E1 -1695.766,E2 -1695.766} C_VEL
LIN {X 0,Y 580.061,Z 432.816,A -85,B 0,C 180,E1 -1696.692,E2 -1696.692} C_VEL
LIN {X 0,Y 580.05,Z 432.217,A -85,B 0,C 180,E1 -1697.404,E2 -1697.404} C_VEL
LIN {X 0,Y 580.054,Z 431.222,A -85,B 0,C 180,E1 -1698.114,E2 -1698.114} C_VEL
LIN {X 0,Y 580.076,Z 429.549,A -85,B 0,C 180,E1 -1698.925,E2 -1698.925} C_VEL
LIN {X 0,Y 580.083,Z 425.606,A -85,B 0,C 180,E1 -1700.235,E2 -1700.235} C_VEL
LIN {X 0,Y 580.113,Z 421.224,A -85,B 0,C 180,E1 -1701.291,E2 -1701.291} C_VEL
LIN {X 0,Y 580.155,Z 414.594,A -85,B 0,C 180,E1 -1702.518,E2 -1702.518} C_VEL
LIN {X 0,Y 580.199,Z 407.27,A -85,B 0,C 180,E1 -1703.583,E2 -1703.583} C_VEL
LIN {X 0,Y 580.288,Z 398.447,A -85,B 0,C 180,E1 -1704.615,E2 -1704.615} C_VEL
LIN {X 0,Y 580.317,Z 388.24,A -85,B 0,C 180,E1 -1705.573,E2 -1705.573} C_VEL
LIN {X 0,Y 580.407,Z 377.89,A -85,B 0,C 180,E1 -1706.356,E2 -1706.356} C_VEL
LIN {X 0,Y 580.536,Z 366.337,A -85,B 0,C 180,E1 -1707.052,E2 -1707.052} C_VEL
LIN {X 0,Y 580.614,Z 354.237,A -85,B 0,C 180,E1 -1707.616,E2 -1707.616} C_VEL
LIN {X 0,Y 580.671,Z 341.558,A -85,B 0,C 180,E1 -1708.05,E2 -1708.05} C_VEL
LIN {X 0,Y 580.759,Z 327.981,A -85,B 0,C 180,E1 -1708.354,E2 -1708.354} C_VEL
LIN {X 0,Y 580.825,Z 225.973,A -85,B 0,C 180,E1 -1709.632,E2 -1709.632} C_VEL
LIN {X 0,Y 580.266,Z 222.606,A -85,B 0,C 180,E1 -1709.697,E2 -1709.697} C_VEL
LIN {X 0,Y 580.353,Z 209.591,A -85,B 0,C 180,E1 -1712.083,E2 -1712.083} C_VEL
LIN {X 0,Y 580.377,Z 198.35,A -85,B 0,C 180,E1 -1714.167,E2 -1714.167} C_VEL
LIN {X 0,Y 580.266,Z 197.203,A -85,B 0,C 180,E1 -1714.429,E2 -1714.429} C_VEL
LIN {X 0,Y 580.333,Z 197.194,A -85,B 0,C 180,E1 -1716.956,E2 -1716.956} C_VEL
LIN {X 0,Y 580.256,Z 197.204,A -85,B 0,C 180,E1 -1719.763,E2 -1719.763} C_VEL
LIN {X 0,Y 580.306,Z 197.196,A -85,B 0,C 180,E1 -1721.882,E2 -1721.882} C_VEL
LIN {X 0,Y 580.276,Z 197.201,A -85,B 0,C 180,E1 -1724.735,E2 -1724.735} C_VEL
LIN {X 0,Y 580.267,Z 197.202,A -85,B 0,C 180,E1 -1727.626,E2 -1727.626} C_VEL
LIN {X 0,Y 580.283,Z 197.198,A -85,B 0,C 180,E1 -1729.824,E2 -1729.824} C_VEL
LIN {X 0,Y 580.254,Z 197.201,A -85,B 0,C 180,E1 -1732.054,E2 -1732.054} C_VEL
LIN {X 0,Y 580.261,Z 197.207,A -85,B 0,C 180,E1 -1734.716,E2 -1734.716} C_VEL
LIN {X 0,Y 580.25,Z 197.204,A -85,B 0,C 180,E1 -1737.404,E2 -1737.404} C_VEL
LIN {X 0,Y 580.267,Z 197.2,A -85,B 0,C 180,E1 -1739.775,E2 -1739.775} C_VEL
LIN {X 0,Y 580.293,Z 197.199,A -85,B 0,C 180,E1 -1742.202,E2 -1742.202} C_VEL
LIN {X 0,Y 580.274,Z 197.207,A -85,B 0,C 180,E1 -1744.698,E2 -1744.698} C_VEL
LIN {X 0,Y 580.269,Z 197.2,A -85,B 0,C 180,E1 -1747.271,E2 -1747.271} C_VEL
LIN {X 0,Y 580.27,Z 197.201,A -85,B 0,C 180,E1 -1749.936,E2 -1749.936} C_VEL
LIN {X 0,Y 580.254,Z 197.206,A -85,B 0,C 180,E1 -1752.709,E2 -1752.709} C_VEL
LIN {X 0,Y 580.241,Z 197.204,A -85,B 0,C 180,E1 -1755.613,E2 -1755.613} C_VEL
LIN {X 0,Y 580.236,Z 197.212,A -85,B 0,C 180,E1 -1758.227,E2 -1758.227} C_VEL
LIN {X 0,Y 580.238,Z 197.203,A -85,B 0,C 180,E1 -1760.961,E2 -1760.961} C_VEL
LIN {X 0,Y 580.211,Z 197.209,A -85,B 0,C 180,E1 -1763.592,E2 -1763.592} C_VEL
LIN {X 0,Y 580.261,Z 197.208,A -85,B 0,C 180,E1 -1766.141,E2 -1766.141} C_VEL
LIN {X 0,Y 580.243,Z 197.204,A -85,B 0,C 180,E1 -1768.612,E2 -1768.612} C_VEL
LIN {X 0,Y 580.246,Z 197.202,A -85,B 0,C 180,E1 -1771.021,E2 -1771.021} C_VEL
LIN {X 0,Y 580.249,Z 197.21,A -85,B 0,C 180,E1 -1773.676,E2 -1773.676} C_VEL
LIN {X 0,Y 580.265,Z 197.201,A -85,B 0,C 180,E1 -1776.441,E2 -1776.441} C_VEL
LIN {X 0,Y 580.269,Z 197.206,A -85,B 0,C 180,E1 -1779.437,E2 -1779.437} C_VEL
LIN {X 0,Y 580.297,Z 197.293,A -85,B 0,C 180,E1 -1780.723,E2 -1780.723} C_VEL
LIN {X 0,Y 580.396,Z 210.114,A -85,B 0,C 180,E1 -1783.105,E2 -1783.105} C_VEL
LIN {X 0,Y 580.295,Z 222.619,A -85,B 0,C 180,E1 -1785.396,E2 -1785.396} C_VEL
LIN {X 0,Y 580.973,Z 228.287,A -85,B 0,C 180,E1 -1785.49,E2 -1785.49} C_VEL
LIN {X 0,Y 580.784,Z 328.72,A -85,B 0,C 180,E1 -1786.752,E2 -1786.752} C_VEL
LIN {X 0,Y 580.759,Z 341.525,A -85,B 0,C 180,E1 -1787.041,E2 -1787.041} C_VEL
LIN {X 0,Y 580.667,Z 353.809,A -85,B 0,C 180,E1 -1787.461,E2 -1787.461} C_VEL
LIN {X 0,Y 580.57,Z 364.503,A -85,B 0,C 180,E1 -1787.947,E2 -1787.947} C_VEL
LIN {X 0,Y 580.462,Z 375.305,A -85,B 0,C 180,E1 -1788.565,E2 -1788.565} C_VEL
LIN {X 0,Y 580.384,Z 386.397,A -85,B 0,C 180,E1 -1789.367,E2 -1789.367} C_VEL
LIN {X 0,Y 580.274,Z 396.068,A -85,B 0,C 180,E1 -1790.237,E2 -1790.237} C_VEL
LIN {X 0,Y 580.226,Z 404.097,A -85,B 0,C 180,E1 -1791.116,E2 -1791.116} C_VEL
LIN {X 0,Y 580.166,Z 412.008,A -85,B 0,C 180,E1 -1792.167,E2 -1792.167} C_VEL
LIN {X 0,Y 580.121,Z 419.357,A -85,B 0,C 180,E1 -1793.421,E2 -1793.421} C_VEL
LIN {X 0,Y 580.129,Z 423.99,A -85,B 0,C 180,E1 -1794.438,E2 -1794.438} C_VEL
LIN {X 0,Y 580.107,Z 427.663,A -85,B 0,C 180,E1 -1795.483,E2 -1795.483} C_VEL
LIN {X 0,Y 580.109,Z 430.336,A -85,B 0,C 180,E1 -1796.527,E2 -1796.527} C_VEL
LIN {X 0,Y 580.042,Z 431.622,A -85,B 0,C 180,E1 -1797.222,E2 -1797.222} C_VEL
LIN {X 0,Y 580.036,Z 432.47,A -85,B 0,C 180,E1 -1797.917,E2 -1797.917} C_VEL
LIN {X 0,Y 580.04,Z 432.948,A -85,B 0,C 180,E1 -1799.306,E2 -1799.306} C_VEL
LIN {X 0,Y 580.038,Z 432.615,A -85,B 0,C 180,E1 -1800,E2 -1800} C_VEL
LIN {X 0,Y 580.049,Z 430.7,A -85,B 0,C 180,E1 -1801.388,E2 -1801.388} C_VEL
LIN {X 0,Y 580.103,Z 428.192,A -85,B 0,C 180,E1 -1802.43,E2 -1802.43} C_VEL
LIN {X 0,Y 580.126,Z 424.693,A -85,B 0,C 180,E1 -1803.473,E2 -1803.473} C_VEL
LIN {X 0,Y 580.126,Z 420.108,A -85,B 0,C 180,E1 -1804.516,E2 -1804.516} C_VEL
LIN {X 0,Y 580.175,Z 413.225,A -85,B 0,C 180,E1 -1805.735,E2 -1805.735} C_VEL
LIN {X 0,Y 580.227,Z 405.513,A -85,B 0,C 180,E1 -1806.806,E2 -1806.806} C_VEL
LIN {X 0,Y 580.266,Z 398.021,A -85,B 0,C 180,E1 -1807.656,E2 -1807.656} C_VEL
LIN {X 0,Y 580.36,Z 388.681,A -85,B 0,C 180,E1 -1808.531,E2 -1808.531} C_VEL
LIN {X 0,Y 580.439,Z 378.395,A -85,B 0,C 180,E1 -1809.32,E2 -1809.32} C_VEL
LIN {X 0,Y 580.57,Z 366.911,A -85,B 0,C 180,E1 -1810.021,E2 -1810.021} C_VEL
LIN {X 0,Y 580.635,Z 354.711,A -85,B 0,C 180,E1 -1810.593,E2 -1810.593} C_VEL
LIN {X 0,Y 580.709,Z 342.132,A -85,B 0,C 180,E1 -1811.033,E2 -1811.033} C_VEL
LIN {X 0,Y 580.76,Z 328.916,A -85,B 0,C 180,E1 -1811.335,E2 -1811.335} C_VEL
LIN {X 0,Y 580.887,Z 226.627,A -85,B 0,C 180,E1 -1812.623,E2 -1812.623} C_VEL
LIN {X 0,Y 580.24,Z 222.573,A -85,B 0,C 180,E1 -1812.704,E2 -1812.704} C_VEL
LIN {X 0,Y 580.376,Z 207.596,A -85,B 0,C 180,E1 -1815.45,E2 -1815.45} C_VEL
LIN {X 0,Y 580.344,Z 197.194,A -85,B 0,C 180,E1 -1817.398,E2 -1817.398} C_VEL
LIN {X 0,Y 580.291,Z 197.199,A -85,B 0,C 180,E1 -1819.823,E2 -1819.823} C_VEL
LIN {X 0,Y 580.273,Z 197.203,A -85,B 0,C 180,E1 -1822.053,E2 -1822.053} C_VEL
LIN {X 0,Y 580.305,Z 197.196,A -85,B 0,C 180,E1 -1825.08,E2 -1825.08} C_VEL
LIN {X 0,Y 580.301,Z 197.203,A -85,B 0,C 180,E1 -1828.185,E2 -1828.185} C_VEL
LIN {X 0,Y 580.28,Z 197.202,A -85,B 0,C 180,E1 -1830.693,E2 -1830.693} C_VEL
LIN {X 0,Y 580.288,Z 197.197,A -85,B 0,C 180,E1 -1833.313,E2 -1833.313} C_VEL
LIN {X 0,Y 580.249,Z 197.204,A -85,B 0,C 180,E1 -1835.756,E2 -1835.756} C_VEL
LIN {X 0,Y 580.292,Z 197.205,A -85,B 0,C 180,E1 -1838.146,E2 -1838.146} C_VEL
LIN {X 0,Y 580.3,Z 197.196,A -85,B 0,C 180,E1 -1840.843,E2 -1840.843} C_VEL
LIN {X 0,Y 580.274,Z 197.201,A -85,B 0,C 180,E1 -1843.658,E2 -1843.658} C_VEL
LIN {X 0,Y 580.272,Z 197.201,A -85,B 0,C 180,E1 -1846.61,E2 -1846.61} C_VEL
LIN {X 0,Y 580.3,Z 197.195,A -85,B 0,C 180,E1 -1849.156,E2 -1849.156} C_VEL
LIN {X 0,Y 580.291,Z 197.205,A -85,B 0,C 180,E1 -1851.927,E2 -1851.927} C_VEL
LIN {X 0,Y 580.252,Z 197.204,A -85,B 0,C 180,E1 -1854.452,E2 -1854.452} C_VEL
LIN {X 0,Y 580.293,Z 197.197,A -85,B 0,C 180,E1 -1856.975,E2 -1856.975} C_VEL
LIN {X 0,Y 580.298,Z 197.2,A -85,B 0,C 180,E1 -1859.424,E2 -1859.424} C_VEL
LIN {X 0,Y 580.263,Z 197.206,A -85,B 0,C 180,E1 -1862.148,E2 -1862.148} C_VEL
LIN {X 0,Y 580.326,Z 197.196,A -85,B 0,C 180,E1 -1865.269,E2 -1865.269} C_VEL
LIN {X 0,Y 580.317,Z 197.353,A -85,B 0,C 180,E1 -1866.301,E2 -1866.301} C_VEL
LIN {X 0,Y 580.942,Z 201.906,A -85,B 0,C 180,E1 -1866.951,E2 -1866.951} C_VEL
LIN {X 0,Y 580.833,Z 220.074,A -85,B 0,C 180,E1 -1869.457,E2 -1869.457} C_VEL
LIN {X 0,Y 580.621,Z 241.348,A -85,B 0,C 180,E1 -1872.385,E2 -1872.385} C_VEL
LIN {X 0,Y 580.458,Z 261.292,A -85,B 0,C 180,E1 -1875.09,E2 -1875.09} C_VEL
LIN {X 0,Y 580.396,Z 270.516,A -85,B 0,C 180,E1 -1876.33,E2 -1876.33} C_VEL
LIN {X 0,Y 580.935,Z 276.45,A -85,B 0,C 180,E1 -1876.421,E2 -1876.421} C_VEL
LIN {X 0,Y 580.811,Z 378.907,A -85,B 0,C 180,E1 -1877.708,E2 -1877.708} C_VEL
LIN {X 0,Y 580.739,Z 392.188,A -85,B 0,C 180,E1 -1878.016,E2 -1878.016} C_VEL
LIN {X 0,Y 580.657,Z 405.126,A -85,B 0,C 180,E1 -1878.466,E2 -1878.466} C_VEL
LIN {X 0,Y 580.554,Z 416.616,A -85,B 0,C 180,E1 -1879.008,E2 -1879.008} C_VEL
LIN {X 0,Y 580.443,Z 428.191,A -85,B 0,C 180,E1 -1879.711,E2 -1879.711} C_VEL
LIN {X 0,Y 580.345,Z 438.591,A -85,B 0,C 180,E1 -1880.502,E2 -1880.502} C_VEL
LIN {X 0,Y 580.272,Z 447.105,A -85,B 0,C 180,E1 -1881.292,E2 -1881.292} C_VEL
LIN {X 0,Y 580.222,Z 454.954,A -85,B 0,C 180,E1 -1882.167,E2 -1882.167} C_VEL
LIN {X 0,Y 580.154,Z 462.647,A -85,B 0,C 180,E1 -1883.221,E2 -1883.221} C_VEL
LIN {X 0,Y 580.139,Z 469.676,A -85,B 0,C 180,E1 -1884.438,E2 -1884.438} C_VEL
LIN {X 0,Y 580.108,Z 474.368,A -85,B 0,C 180,E1 -1885.483,E2 -1885.483} C_VEL
LIN {X 0,Y 580.123,Z 477.956,A -85,B 0,C 180,E1 -1886.527,E2 -1886.527} C_VEL
LIN {X 0,Y 580.043,Z 479.808,A -85,B 0,C 180,E1 -1887.221,E2 -1887.221} C_VEL
LIN {X 0,Y 580.04,Z 481.199,A -85,B 0,C 180,E1 -1887.916,E2 -1887.916} C_VEL
LIN {X 0,Y 580.04,Z 482.784,A -85,B 0,C 180,E1 -1889.305,E2 -1889.305} C_VEL
LIN {X 0,Y 580.037,Z 483,A -85,B 0,C 180,E1 -1889.999,E2 -1889.999} C_VEL
LIN {X 0,Y 580.046,Z 482.186,A -85,B 0,C 180,E1 -1891.388,E2 -1891.388} C_VEL
LIN {X 0,Y 580.04,Z 481.2,A -85,B 0,C 180,E1 -1892.082,E2 -1892.082} C_VEL
LIN {X 0,Y 580.043,Z 479.81,A -85,B 0,C 180,E1 -1892.777,E2 -1892.777} C_VEL
LIN {X 0,Y 580.11,Z 476.898,A -85,B 0,C 180,E1 -1893.82,E2 -1893.82} C_VEL
LIN {X 0,Y 580.053,Z 472.953,A -85,B 0,C 180,E1 -1894.864,E2 -1894.864} C_VEL
LIN {X 0,Y 580.139,Z 466.881,A -85,B 0,C 180,E1 -1896.084,E2 -1896.084} C_VEL
LIN {X 0,Y 580.184,Z 460.243,A -85,B 0,C 180,E1 -1897.132,E2 -1897.132} C_VEL
LIN {X 0,Y 580.25,Z 451.997,A -85,B 0,C 180,E1 -1898.181,E2 -1898.181} C_VEL
LIN {X 0,Y 580.307,Z 443.547,A -85,B 0,C 180,E1 -1899.058,E2 -1899.058} C_VEL
LIN {X 0,Y 580.425,Z 433.109,A -85,B 0,C 180,E1 -1899.935,E2 -1899.935} C_VEL
LIN {X 0,Y 580.492,Z 422.767,A -85,B 0,C 180,E1 -1900.639,E2 -1900.639} C_VEL
LIN {X 0,Y 580.595,Z 411.261,A -85,B 0,C 180,E1 -1901.263,E2 -1901.263} C_VEL
LIN {X 0,Y 580.678,Z 398.502,A -85,B 0,C 180,E1 -1901.784,E2 -1901.784} C_VEL
LIN {X 0,Y 580.777,Z 385.472,A -85,B 0,C 180,E1 -1902.159,E2 -1902.159} C_VEL
LIN {X 0,Y 580.852,Z 373.145,A -85,B 0,C 180,E1 -1902.379,E2 -1902.379} C_VEL
LIN {X 0,Y 580.809,Z 273.224,A -85,B 0,C 180,E1 -1903.622,E2 -1903.622} C_VEL
LIN {X 0,Y 580.415,Z 270.445,A -85,B 0,C 180,E1 -1903.679,E2 -1903.679} C_VEL
LIN {X 0,Y 580.597,Z 248.008,A -85,B 0,C 180,E1 -1906.707,E2 -1906.707} C_VEL
LIN {X 0,Y 580.778,Z 226.594,A -85,B 0,C 180,E1 -1909.64,E2 -1909.64} C_VEL
LIN {X 0,Y 580.943,Z 206.683,A -85,B 0,C 180,E1 -1912.399,E2 -1912.399} C_VEL
LIN {X 0,Y 580.898,Z 200.296,A -85,B 0,C 180,E1 -1913.289,E2 -1913.289} C_VEL
LIN {X 0,Y 580.282,Z 197.206,A -85,B 0,C 180,E1 -1913.746,E2 -1913.746} C_VEL
LIN {X 0,Y 580.281,Z 197.205,A -85,B 0,C 180,E1 -1916.331,E2 -1916.331} C_VEL
LIN {X 0,Y 580.295,Z 197.197,A -85,B 0,C 180,E1 -1919.308,E2 -1919.308} C_VEL
LIN {X 0,Y 580.291,Z 197.199,A -85,B 0,C 180,E1 -1922.2,E2 -1922.2} C_VEL
LIN {X 0,Y 580.281,Z 197.196,A -85,B 0,C 180,E1 -1924.696,E2 -1924.696} C_VEL
LIN {X 0,Y 580.282,Z 197.2,A -85,B 0,C 180,E1 -1927.268,E2 -1927.268} C_VEL
LIN {X 0,Y 580.28,Z 197.199,A -85,B 0,C 180,E1 -1930.269,E2 -1930.269} C_VEL
LIN {X 0,Y 580.253,Z 197.2,A -85,B 0,C 180,E1 -1932.707,E2 -1932.707} C_VEL
LIN {X 0,Y 580.243,Z 197.211,A -85,B 0,C 180,E1 -1935.61,E2 -1935.61} C_VEL
LIN {X 0,Y 580.25,Z 197.2,A -85,B 0,C 180,E1 -1938.228,E2 -1938.228} C_VEL
LIN {X 0,Y 580.259,Z 197.203,A -85,B 0,C 180,E1 -1940.963,E2 -1940.963} C_VEL
LIN {X 0,Y 580.258,Z 197.203,A -85,B 0,C 180,E1 -1943.596,E2 -1943.596} C_VEL
LIN {X 0,Y 580.268,Z 197.198,A -85,B 0,C 180,E1 -1946.142,E2 -1946.142} C_VEL
LIN {X 0,Y 580.255,Z 197.202,A -85,B 0,C 180,E1 -1948.613,E2 -1948.613} C_VEL
LIN {X 0,Y 580.269,Z 197.205,A -85,B 0,C 180,E1 -1951.023,E2 -1951.023} C_VEL
LIN {X 0,Y 580.244,Z 197.203,A -85,B 0,C 180,E1 -1953.673,E2 -1953.673} C_VEL
LIN {X 0,Y 580.234,Z 197.204,A -85,B 0,C 180,E1 -1956.44,E2 -1956.44} C_VEL
LIN {X 0,Y 580.24,Z 197.203,A -85,B 0,C 180,E1 -1959.436,E2 -1959.436} C_VEL
LIN {X 0,Y 580.225,Z 197.204,A -85,B 0,C 180,E1 -1961.644,E2 -1961.644} C_VEL
LIN {X 0,Y 580.231,Z 197.203,A -85,B 0,C 180,E1 -1963.824,E2 -1963.824} C_VEL
LIN {X 0,Y 580.271,Z 197.196,A -85,B 0,C 180,E1 -1965.982,E2 -1965.982} C_VEL
LIN {X 0,Y 580.296,Z 197.201,A -85,B 0,C 180,E1 -1968.827,E2 -1968.827} C_VEL
LIN {X 0,Y 580.278,Z 197.198,A -85,B 0,C 180,E1 -1971.643,E2 -1971.643} C_VEL
LIN {X 0,Y 580.302,Z 197.201,A -85,B 0,C 180,E1 -1974.44,E2 -1974.44} C_VEL
LIN {X 0,Y 580.305,Z 197.194,A -85,B 0,C 180,E1 -1977.223,E2 -1977.223} C_VEL
LIN {X 0,Y 580.333,Z 197.196,A -85,B 0,C 180,E1 -1980,E2 -1980} C_VEL
LIN {X 0,Y 580.32,Z 197.191,A -85,B 0,C 180,E1 -1982.777,E2 -1982.777} C_VEL
LIN {X 0,Y 580.295,Z 197.197,A -85,B 0,C 180,E1 -1985.56,E2 -1985.56} C_VEL
LIN {X 0,Y 580.306,Z 197.197,A -85,B 0,C 180,E1 -1987.656,E2 -1987.656} C_VEL
LIN {X 0,Y 580.286,Z 197.197,A -85,B 0,C 180,E1 -1990.467,E2 -1990.467} C_VEL
LIN {X 0,Y 580.256,Z 197.201,A -85,B 0,C 180,E1 -1993.305,E2 -1993.305} C_VEL
LIN {X 0,Y 580.281,Z 197.201,A -85,B 0,C 180,E1 -1995.453,E2 -1995.453} C_VEL
LIN {X 0,Y 580.279,Z 197.203,A -85,B 0,C 180,E1 -1997.625,E2 -1997.625} C_VEL
